// TIA Portal V16 export
// export: Created 2024-09-05T17:39:09.6685923Z, ExportSetting WithDefaults, DisplayName Totally Integrated Automation Portal, DisplayVersion V16 Update 6, DisplayName TIA Portal Version Control Interface, DisplayVersion V16 Update 2, DisplayName TIA Portal Openness, DisplayVersion V16 Update 6, DisplayName STEP 7 Professional, DisplayVersion V16 Update 6, DisplayName STEP 7 Safety, DisplayVersion V16, DisplayName WinCC Advanced, DisplayVersion V16 Update 6
DATA_BLOCK "CylinderGeneratedCalls_DB"   // DB51
VERSION : 0.1
// stored: AutoNumber true, DBAccessibleFromOPCUA true, InstanceOfName CylinderGeneratedCalls, InstanceOfType FB
"CylinderGeneratedCalls"
   // VAR
   //    MM2200_GrippingTubeFrontInstant { S7_SetPoint := 'True'} : "CylinderFaceplate";
   //    MM2201_GrippingTubeRearInstant { S7_SetPoint := 'True'} : "CylinderFaceplate";
   //    MM2220_HoldingSidememberInsideLeftInstant { S7_SetPoint := 'True'} : "CylinderFaceplate";
   //    MM2221_HoldingSidememberInsideRightInstant { S7_SetPoint := 'True'} : "CylinderFaceplate";
   //    MM2240_HoldingSidememberOutsideLeftInstant { S7_SetPoint := 'True'} : "CylinderFaceplate";
   //    MM2241_HoldingSidememberOutsideRightInstant { S7_SetPoint := 'True'} : "CylinderFaceplate";
   //    MM2500_GrippingTubeFrontInstant { S7_SetPoint := 'True'} : "CylinderFaceplate";
   //    MM2501_GrippingTubeRearInstant { S7_SetPoint := 'True'} : "CylinderFaceplate";
   //    MM2520_HoldingSidememberInsideLeftInstant { S7_SetPoint := 'True'} : "CylinderFaceplate";
   //    MM2521_HoldingSidememberInsideRightInstant { S7_SetPoint := 'True'} : "CylinderFaceplate";
   //    MM2540_HoldingSidememberOutsideLeftInstant { S7_SetPoint := 'True'} : "CylinderFaceplate";
   //    MM2541_HoldingSidememberOutsideRightInstant { S7_SetPoint := 'True'} : "CylinderFaceplate";
   //    MM300_ShiftingSupportRightInstant { S7_SetPoint := 'True'} : "CylinderFaceplate";
   //    MM302_ShiftingSupportLeftInstant { S7_SetPoint := 'True'} : "CylinderFaceplate";
   //    MM304_MovingStopRightInstant { S7_SetPoint := 'True'} : "CylinderFaceplate";
   //    MM306_MovingStopLeftInstant { S7_SetPoint := 'True'} : "CylinderFaceplate";
   //    MM340_RivetingUnitRightInstant { S7_SetPoint := 'True'} : "CylinderFaceplate";
   //    MM342_RivetingUnitLeftInstant { S7_SetPoint := 'True'} : "CylinderFaceplate";
   //    MM344_RivetingSupportRightInstant { S7_SetPoint := 'True'} : "CylinderFaceplate";
   //    MM346_RivetingSupportLeftInstant { S7_SetPoint := 'True'} : "CylinderFaceplate";
   //    MM350_ShiftWedgeRightInstant { S7_SetPoint := 'True'} : "CylinderFaceplate";
   //    MM352_ShiftWedgeLeftInstant { S7_SetPoint := 'True'} : "CylinderFaceplate";
   //    MM104_AutoejectGripperLiftingInstant { S7_SetPoint := 'True'} : "CylinderFaceplate";
   //    MM3100_SidememberSupportLeftInstant { S7_SetPoint := 'True'} : "CylinderFaceplate";
   //    MM3101_SidememberSupportRightInstant { S7_SetPoint := 'True'} : "CylinderFaceplate";
   // END_VAR
BEGIN
   MM2200_GrippingTubeFrontInstant.POWER_OK := TRUE;
   MM2200_GrippingTubeFrontInstant.CylinderNumber := 0;
   MM2200_GrippingTubeFrontInstant.HMICommand := 0;
   MM2200_GrippingTubeFrontInstant.BasicPositionCondition := TRUE;
   MM2200_GrippingTubeFrontInstant.WorkPositionCondition := FALSE;
   MM2200_GrippingTubeFrontInstant.BasicPositionSensor := TRUE;
   MM2200_GrippingTubeFrontInstant.WorkPositionSensor := FALSE;
   MM2200_GrippingTubeFrontInstant.TRIGGER := TRUE;
   MM2200_GrippingTubeFrontInstant.RESET := FALSE;
   MM2200_GrippingTubeFrontInstant.DELAY_BASIC := T#100MS;
   MM2200_GrippingTubeFrontInstant.DELAY_WORK := T#100MS;
   MM2200_GrippingTubeFrontInstant.DELAY_FREE := T#100MS;
   MM2200_GrippingTubeFrontInstant.ERROR_TIME := T#10S;
   MM2200_GrippingTubeFrontInstant.ValveDelay := T#0MS;
   MM2200_GrippingTubeFrontInstant.iNoCollisionBasic := TRUE;
   MM2200_GrippingTubeFrontInstant.iNoCollisionWork := TRUE;
   MM2200_GrippingTubeFrontInstant.iNoCollisionFree := TRUE;
   MM2200_GrippingTubeFrontInstant.VALVE_BASIC := TRUE;
   MM2200_GrippingTubeFrontInstant.VALVE_WORK := FALSE;
   MM2200_GrippingTubeFrontInstant.ERROR_BASIC := FALSE;
   MM2200_GrippingTubeFrontInstant.ERROR_WORK := FALSE;
   MM2200_GrippingTubeFrontInstant.HMIStatus := 257;
   MM2200_GrippingTubeFrontInstant.MOVE_BASIC := TRUE;
   MM2200_GrippingTubeFrontInstant.MOVE_WORK := FALSE;
   MM2200_GrippingTubeFrontInstant.MOVE_FREE := FALSE;
   MM2200_GrippingTubeFrontInstant."4l+Started" := FALSE;
   MM2200_GrippingTubeFrontInstant.InitCommandBP := FALSE;
   MM2200_GrippingTubeFrontInstant.InitCommandWP := FALSE;
   MM2200_GrippingTubeFrontInstant.BasicWorkStartWP := FALSE;
   MM2200_GrippingTubeFrontInstant.BasicWorkStartBP := FALSE;
   MM2200_GrippingTubeFrontInstant.work_valve := FALSE;
   MM2200_GrippingTubeFrontInstant.basic_valve := TRUE;
   MM2200_GrippingTubeFrontInstant.free_valve := FALSE;
   MM2200_GrippingTubeFrontInstant.baspos_error.PT := T#10S;
   MM2200_GrippingTubeFrontInstant.baspos_error.IN := FALSE;
   MM2200_GrippingTubeFrontInstant.workpos_error.PT := T#10S;
   MM2200_GrippingTubeFrontInstant.workpos_error.IN := FALSE;
   MM2200_GrippingTubeFrontInstant.baspos_delay.PT := T#100MS;
   MM2200_GrippingTubeFrontInstant.baspos_delay.IN := TRUE;
   MM2200_GrippingTubeFrontInstant.workpos_delay.PT := T#100MS;
   MM2200_GrippingTubeFrontInstant.workpos_delay.IN := FALSE;
   MM2200_GrippingTubeFrontInstant.CylinderOperationOld.InWp := FALSE;
   MM2200_GrippingTubeFrontInstant.CylinderOperationOld.InBp := TRUE;
   MM2200_GrippingTubeFrontInstant.CylinderOperationOld.InFp := FALSE;
   MM2200_GrippingTubeFrontInstant.CylinderOperationOld.ToWp := FALSE;
   MM2200_GrippingTubeFrontInstant.CylinderOperationOld.ToBp := TRUE;
   MM2200_GrippingTubeFrontInstant.CylinderOperationOld.ToFp := FALSE;
   MM2200_GrippingTubeFrontInstant.IEC_Timer_0_Instance.PT := T#0MS;
   MM2200_GrippingTubeFrontInstant.IEC_Timer_0_Instance.IN := FALSE;
   MM2200_GrippingTubeFrontInstant.R_TRIG_Instance.CLK := FALSE;
   MM2200_GrippingTubeFrontInstant.R_TRIG_Instance.Q := FALSE;
   MM2200_GrippingTubeFrontInstant.R_TRIG_Instance.Stat_Bit := FALSE;
   MM2200_GrippingTubeFrontInstant.IEC_Timer_0_Instance_1.PT := T#0MS;
   MM2200_GrippingTubeFrontInstant.IEC_Timer_0_Instance_1.IN := FALSE;
   MM2200_GrippingTubeFrontInstant.IEC_Timer_0_Instance_2.PT := T#0MS;
   MM2200_GrippingTubeFrontInstant.IEC_Timer_0_Instance_2.IN := FALSE;
   MM2200_GrippingTubeFrontInstant.IEC_Timer_0_Instance_3.PT := T#0MS;
   MM2200_GrippingTubeFrontInstant.IEC_Timer_0_Instance_3.IN := FALSE;
   MM2200_GrippingTubeFrontInstant.IEC_Timer_0_Instance_4.PT := T#0MS;
   MM2200_GrippingTubeFrontInstant.IEC_Timer_0_Instance_4.IN := TRUE;
   MM2201_GrippingTubeRearInstant.POWER_OK := TRUE;
   MM2201_GrippingTubeRearInstant.CylinderNumber := 1;
   MM2201_GrippingTubeRearInstant.HMICommand := 0;
   MM2201_GrippingTubeRearInstant.BasicPositionCondition := TRUE;
   MM2201_GrippingTubeRearInstant.WorkPositionCondition := FALSE;
   MM2201_GrippingTubeRearInstant.BasicPositionSensor := TRUE;
   MM2201_GrippingTubeRearInstant.WorkPositionSensor := FALSE;
   MM2201_GrippingTubeRearInstant.TRIGGER := TRUE;
   MM2201_GrippingTubeRearInstant.RESET := FALSE;
   MM2201_GrippingTubeRearInstant.DELAY_BASIC := T#100MS;
   MM2201_GrippingTubeRearInstant.DELAY_WORK := T#100MS;
   MM2201_GrippingTubeRearInstant.DELAY_FREE := T#100MS;
   MM2201_GrippingTubeRearInstant.ERROR_TIME := T#10S;
   MM2201_GrippingTubeRearInstant.ValveDelay := T#0MS;
   MM2201_GrippingTubeRearInstant.iNoCollisionBasic := TRUE;
   MM2201_GrippingTubeRearInstant.iNoCollisionWork := TRUE;
   MM2201_GrippingTubeRearInstant.iNoCollisionFree := TRUE;
   MM2201_GrippingTubeRearInstant.VALVE_BASIC := TRUE;
   MM2201_GrippingTubeRearInstant.VALVE_WORK := FALSE;
   MM2201_GrippingTubeRearInstant.ERROR_BASIC := FALSE;
   MM2201_GrippingTubeRearInstant.ERROR_WORK := FALSE;
   MM2201_GrippingTubeRearInstant.HMIStatus := 257;
   MM2201_GrippingTubeRearInstant.MOVE_BASIC := TRUE;
   MM2201_GrippingTubeRearInstant.MOVE_WORK := FALSE;
   MM2201_GrippingTubeRearInstant.MOVE_FREE := FALSE;
   MM2201_GrippingTubeRearInstant."4l+Started" := FALSE;
   MM2201_GrippingTubeRearInstant.InitCommandBP := FALSE;
   MM2201_GrippingTubeRearInstant.InitCommandWP := FALSE;
   MM2201_GrippingTubeRearInstant.BasicWorkStartWP := FALSE;
   MM2201_GrippingTubeRearInstant.BasicWorkStartBP := FALSE;
   MM2201_GrippingTubeRearInstant.work_valve := FALSE;
   MM2201_GrippingTubeRearInstant.basic_valve := TRUE;
   MM2201_GrippingTubeRearInstant.free_valve := FALSE;
   MM2201_GrippingTubeRearInstant.baspos_error.PT := T#10S;
   MM2201_GrippingTubeRearInstant.baspos_error.IN := FALSE;
   MM2201_GrippingTubeRearInstant.workpos_error.PT := T#10S;
   MM2201_GrippingTubeRearInstant.workpos_error.IN := FALSE;
   MM2201_GrippingTubeRearInstant.baspos_delay.PT := T#100MS;
   MM2201_GrippingTubeRearInstant.baspos_delay.IN := TRUE;
   MM2201_GrippingTubeRearInstant.workpos_delay.PT := T#100MS;
   MM2201_GrippingTubeRearInstant.workpos_delay.IN := FALSE;
   MM2201_GrippingTubeRearInstant.CylinderOperationOld.InWp := FALSE;
   MM2201_GrippingTubeRearInstant.CylinderOperationOld.InBp := TRUE;
   MM2201_GrippingTubeRearInstant.CylinderOperationOld.InFp := FALSE;
   MM2201_GrippingTubeRearInstant.CylinderOperationOld.ToWp := FALSE;
   MM2201_GrippingTubeRearInstant.CylinderOperationOld.ToBp := TRUE;
   MM2201_GrippingTubeRearInstant.CylinderOperationOld.ToFp := FALSE;
   MM2201_GrippingTubeRearInstant.IEC_Timer_0_Instance.PT := T#0MS;
   MM2201_GrippingTubeRearInstant.IEC_Timer_0_Instance.IN := FALSE;
   MM2201_GrippingTubeRearInstant.R_TRIG_Instance.CLK := FALSE;
   MM2201_GrippingTubeRearInstant.R_TRIG_Instance.Q := FALSE;
   MM2201_GrippingTubeRearInstant.R_TRIG_Instance.Stat_Bit := FALSE;
   MM2201_GrippingTubeRearInstant.IEC_Timer_0_Instance_1.PT := T#0MS;
   MM2201_GrippingTubeRearInstant.IEC_Timer_0_Instance_1.IN := FALSE;
   MM2201_GrippingTubeRearInstant.IEC_Timer_0_Instance_2.PT := T#0MS;
   MM2201_GrippingTubeRearInstant.IEC_Timer_0_Instance_2.IN := FALSE;
   MM2201_GrippingTubeRearInstant.IEC_Timer_0_Instance_3.PT := T#0MS;
   MM2201_GrippingTubeRearInstant.IEC_Timer_0_Instance_3.IN := FALSE;
   MM2201_GrippingTubeRearInstant.IEC_Timer_0_Instance_4.PT := T#0MS;
   MM2201_GrippingTubeRearInstant.IEC_Timer_0_Instance_4.IN := TRUE;
   MM2220_HoldingSidememberInsideLeftInstant.POWER_OK := TRUE;
   MM2220_HoldingSidememberInsideLeftInstant.CylinderNumber := 2;
   MM2220_HoldingSidememberInsideLeftInstant.HMICommand := 0;
   MM2220_HoldingSidememberInsideLeftInstant.BasicPositionCondition := TRUE;
   MM2220_HoldingSidememberInsideLeftInstant.WorkPositionCondition := FALSE;
   MM2220_HoldingSidememberInsideLeftInstant.BasicPositionSensor := TRUE;
   MM2220_HoldingSidememberInsideLeftInstant.WorkPositionSensor := FALSE;
   MM2220_HoldingSidememberInsideLeftInstant.TRIGGER := TRUE;
   MM2220_HoldingSidememberInsideLeftInstant.RESET := FALSE;
   MM2220_HoldingSidememberInsideLeftInstant.DELAY_BASIC := T#100MS;
   MM2220_HoldingSidememberInsideLeftInstant.DELAY_WORK := T#100MS;
   MM2220_HoldingSidememberInsideLeftInstant.DELAY_FREE := T#100MS;
   MM2220_HoldingSidememberInsideLeftInstant.ERROR_TIME := T#10S;
   MM2220_HoldingSidememberInsideLeftInstant.ValveDelay := T#0MS;
   MM2220_HoldingSidememberInsideLeftInstant.iNoCollisionBasic := TRUE;
   MM2220_HoldingSidememberInsideLeftInstant.iNoCollisionWork := TRUE;
   MM2220_HoldingSidememberInsideLeftInstant.iNoCollisionFree := TRUE;
   MM2220_HoldingSidememberInsideLeftInstant.VALVE_BASIC := TRUE;
   MM2220_HoldingSidememberInsideLeftInstant.VALVE_WORK := FALSE;
   MM2220_HoldingSidememberInsideLeftInstant.ERROR_BASIC := FALSE;
   MM2220_HoldingSidememberInsideLeftInstant.ERROR_WORK := FALSE;
   MM2220_HoldingSidememberInsideLeftInstant.HMIStatus := 257;
   MM2220_HoldingSidememberInsideLeftInstant.MOVE_BASIC := TRUE;
   MM2220_HoldingSidememberInsideLeftInstant.MOVE_WORK := FALSE;
   MM2220_HoldingSidememberInsideLeftInstant.MOVE_FREE := FALSE;
   MM2220_HoldingSidememberInsideLeftInstant."4l+Started" := FALSE;
   MM2220_HoldingSidememberInsideLeftInstant.InitCommandBP := FALSE;
   MM2220_HoldingSidememberInsideLeftInstant.InitCommandWP := FALSE;
   MM2220_HoldingSidememberInsideLeftInstant.BasicWorkStartWP := FALSE;
   MM2220_HoldingSidememberInsideLeftInstant.BasicWorkStartBP := FALSE;
   MM2220_HoldingSidememberInsideLeftInstant.work_valve := FALSE;
   MM2220_HoldingSidememberInsideLeftInstant.basic_valve := TRUE;
   MM2220_HoldingSidememberInsideLeftInstant.free_valve := FALSE;
   MM2220_HoldingSidememberInsideLeftInstant.baspos_error.PT := T#10S;
   MM2220_HoldingSidememberInsideLeftInstant.baspos_error.IN := FALSE;
   MM2220_HoldingSidememberInsideLeftInstant.workpos_error.PT := T#10S;
   MM2220_HoldingSidememberInsideLeftInstant.workpos_error.IN := FALSE;
   MM2220_HoldingSidememberInsideLeftInstant.baspos_delay.PT := T#100MS;
   MM2220_HoldingSidememberInsideLeftInstant.baspos_delay.IN := TRUE;
   MM2220_HoldingSidememberInsideLeftInstant.workpos_delay.PT := T#100MS;
   MM2220_HoldingSidememberInsideLeftInstant.workpos_delay.IN := FALSE;
   MM2220_HoldingSidememberInsideLeftInstant.CylinderOperationOld.InWp := FALSE;
   MM2220_HoldingSidememberInsideLeftInstant.CylinderOperationOld.InBp := TRUE;
   MM2220_HoldingSidememberInsideLeftInstant.CylinderOperationOld.InFp := FALSE;
   MM2220_HoldingSidememberInsideLeftInstant.CylinderOperationOld.ToWp := FALSE;
   MM2220_HoldingSidememberInsideLeftInstant.CylinderOperationOld.ToBp := TRUE;
   MM2220_HoldingSidememberInsideLeftInstant.CylinderOperationOld.ToFp := FALSE;
   MM2220_HoldingSidememberInsideLeftInstant.IEC_Timer_0_Instance.PT := T#0MS;
   MM2220_HoldingSidememberInsideLeftInstant.IEC_Timer_0_Instance.IN := FALSE;
   MM2220_HoldingSidememberInsideLeftInstant.R_TRIG_Instance.CLK := FALSE;
   MM2220_HoldingSidememberInsideLeftInstant.R_TRIG_Instance.Q := FALSE;
   MM2220_HoldingSidememberInsideLeftInstant.R_TRIG_Instance.Stat_Bit := FALSE;
   MM2220_HoldingSidememberInsideLeftInstant.IEC_Timer_0_Instance_1.PT := T#0MS;
   MM2220_HoldingSidememberInsideLeftInstant.IEC_Timer_0_Instance_1.IN := FALSE;
   MM2220_HoldingSidememberInsideLeftInstant.IEC_Timer_0_Instance_2.PT := T#0MS;
   MM2220_HoldingSidememberInsideLeftInstant.IEC_Timer_0_Instance_2.IN := FALSE;
   MM2220_HoldingSidememberInsideLeftInstant.IEC_Timer_0_Instance_3.PT := T#0MS;
   MM2220_HoldingSidememberInsideLeftInstant.IEC_Timer_0_Instance_3.IN := FALSE;
   MM2220_HoldingSidememberInsideLeftInstant.IEC_Timer_0_Instance_4.PT := T#0MS;
   MM2220_HoldingSidememberInsideLeftInstant.IEC_Timer_0_Instance_4.IN := TRUE;
   MM2221_HoldingSidememberInsideRightInstant.POWER_OK := TRUE;
   MM2221_HoldingSidememberInsideRightInstant.CylinderNumber := 3;
   MM2221_HoldingSidememberInsideRightInstant.HMICommand := 0;
   MM2221_HoldingSidememberInsideRightInstant.BasicPositionCondition := TRUE;
   MM2221_HoldingSidememberInsideRightInstant.WorkPositionCondition := FALSE;
   MM2221_HoldingSidememberInsideRightInstant.BasicPositionSensor := TRUE;
   MM2221_HoldingSidememberInsideRightInstant.WorkPositionSensor := FALSE;
   MM2221_HoldingSidememberInsideRightInstant.TRIGGER := TRUE;
   MM2221_HoldingSidememberInsideRightInstant.RESET := FALSE;
   MM2221_HoldingSidememberInsideRightInstant.DELAY_BASIC := T#100MS;
   MM2221_HoldingSidememberInsideRightInstant.DELAY_WORK := T#100MS;
   MM2221_HoldingSidememberInsideRightInstant.DELAY_FREE := T#100MS;
   MM2221_HoldingSidememberInsideRightInstant.ERROR_TIME := T#10S;
   MM2221_HoldingSidememberInsideRightInstant.ValveDelay := T#0MS;
   MM2221_HoldingSidememberInsideRightInstant.iNoCollisionBasic := TRUE;
   MM2221_HoldingSidememberInsideRightInstant.iNoCollisionWork := TRUE;
   MM2221_HoldingSidememberInsideRightInstant.iNoCollisionFree := TRUE;
   MM2221_HoldingSidememberInsideRightInstant.VALVE_BASIC := TRUE;
   MM2221_HoldingSidememberInsideRightInstant.VALVE_WORK := FALSE;
   MM2221_HoldingSidememberInsideRightInstant.ERROR_BASIC := FALSE;
   MM2221_HoldingSidememberInsideRightInstant.ERROR_WORK := FALSE;
   MM2221_HoldingSidememberInsideRightInstant.HMIStatus := 257;
   MM2221_HoldingSidememberInsideRightInstant.MOVE_BASIC := TRUE;
   MM2221_HoldingSidememberInsideRightInstant.MOVE_WORK := FALSE;
   MM2221_HoldingSidememberInsideRightInstant.MOVE_FREE := FALSE;
   MM2221_HoldingSidememberInsideRightInstant."4l+Started" := FALSE;
   MM2221_HoldingSidememberInsideRightInstant.InitCommandBP := FALSE;
   MM2221_HoldingSidememberInsideRightInstant.InitCommandWP := FALSE;
   MM2221_HoldingSidememberInsideRightInstant.BasicWorkStartWP := FALSE;
   MM2221_HoldingSidememberInsideRightInstant.BasicWorkStartBP := FALSE;
   MM2221_HoldingSidememberInsideRightInstant.work_valve := FALSE;
   MM2221_HoldingSidememberInsideRightInstant.basic_valve := TRUE;
   MM2221_HoldingSidememberInsideRightInstant.free_valve := FALSE;
   MM2221_HoldingSidememberInsideRightInstant.baspos_error.PT := T#10S;
   MM2221_HoldingSidememberInsideRightInstant.baspos_error.IN := FALSE;
   MM2221_HoldingSidememberInsideRightInstant.workpos_error.PT := T#10S;
   MM2221_HoldingSidememberInsideRightInstant.workpos_error.IN := FALSE;
   MM2221_HoldingSidememberInsideRightInstant.baspos_delay.PT := T#100MS;
   MM2221_HoldingSidememberInsideRightInstant.baspos_delay.IN := TRUE;
   MM2221_HoldingSidememberInsideRightInstant.workpos_delay.PT := T#100MS;
   MM2221_HoldingSidememberInsideRightInstant.workpos_delay.IN := FALSE;
   MM2221_HoldingSidememberInsideRightInstant.CylinderOperationOld.InWp := FALSE;
   MM2221_HoldingSidememberInsideRightInstant.CylinderOperationOld.InBp := TRUE;
   MM2221_HoldingSidememberInsideRightInstant.CylinderOperationOld.InFp := FALSE;
   MM2221_HoldingSidememberInsideRightInstant.CylinderOperationOld.ToWp := FALSE;
   MM2221_HoldingSidememberInsideRightInstant.CylinderOperationOld.ToBp := TRUE;
   MM2221_HoldingSidememberInsideRightInstant.CylinderOperationOld.ToFp := FALSE;
   MM2221_HoldingSidememberInsideRightInstant.IEC_Timer_0_Instance.PT := T#0MS;
   MM2221_HoldingSidememberInsideRightInstant.IEC_Timer_0_Instance.IN := FALSE;
   MM2221_HoldingSidememberInsideRightInstant.R_TRIG_Instance.CLK := FALSE;
   MM2221_HoldingSidememberInsideRightInstant.R_TRIG_Instance.Q := FALSE;
   MM2221_HoldingSidememberInsideRightInstant.R_TRIG_Instance.Stat_Bit := FALSE;
   MM2221_HoldingSidememberInsideRightInstant.IEC_Timer_0_Instance_1.PT := T#0MS;
   MM2221_HoldingSidememberInsideRightInstant.IEC_Timer_0_Instance_1.IN := FALSE;
   MM2221_HoldingSidememberInsideRightInstant.IEC_Timer_0_Instance_2.PT := T#0MS;
   MM2221_HoldingSidememberInsideRightInstant.IEC_Timer_0_Instance_2.IN := FALSE;
   MM2221_HoldingSidememberInsideRightInstant.IEC_Timer_0_Instance_3.PT := T#0MS;
   MM2221_HoldingSidememberInsideRightInstant.IEC_Timer_0_Instance_3.IN := FALSE;
   MM2221_HoldingSidememberInsideRightInstant.IEC_Timer_0_Instance_4.PT := T#0MS;
   MM2221_HoldingSidememberInsideRightInstant.IEC_Timer_0_Instance_4.IN := TRUE;
   MM2240_HoldingSidememberOutsideLeftInstant.POWER_OK := TRUE;
   MM2240_HoldingSidememberOutsideLeftInstant.CylinderNumber := 4;
   MM2240_HoldingSidememberOutsideLeftInstant.HMICommand := 0;
   MM2240_HoldingSidememberOutsideLeftInstant.BasicPositionCondition := TRUE;
   MM2240_HoldingSidememberOutsideLeftInstant.WorkPositionCondition := FALSE;
   MM2240_HoldingSidememberOutsideLeftInstant.BasicPositionSensor := TRUE;
   MM2240_HoldingSidememberOutsideLeftInstant.WorkPositionSensor := FALSE;
   MM2240_HoldingSidememberOutsideLeftInstant.TRIGGER := TRUE;
   MM2240_HoldingSidememberOutsideLeftInstant.RESET := FALSE;
   MM2240_HoldingSidememberOutsideLeftInstant.DELAY_BASIC := T#100MS;
   MM2240_HoldingSidememberOutsideLeftInstant.DELAY_WORK := T#100MS;
   MM2240_HoldingSidememberOutsideLeftInstant.DELAY_FREE := T#100MS;
   MM2240_HoldingSidememberOutsideLeftInstant.ERROR_TIME := T#10S;
   MM2240_HoldingSidememberOutsideLeftInstant.ValveDelay := T#0MS;
   MM2240_HoldingSidememberOutsideLeftInstant.iNoCollisionBasic := TRUE;
   MM2240_HoldingSidememberOutsideLeftInstant.iNoCollisionWork := TRUE;
   MM2240_HoldingSidememberOutsideLeftInstant.iNoCollisionFree := TRUE;
   MM2240_HoldingSidememberOutsideLeftInstant.VALVE_BASIC := TRUE;
   MM2240_HoldingSidememberOutsideLeftInstant.VALVE_WORK := FALSE;
   MM2240_HoldingSidememberOutsideLeftInstant.ERROR_BASIC := FALSE;
   MM2240_HoldingSidememberOutsideLeftInstant.ERROR_WORK := FALSE;
   MM2240_HoldingSidememberOutsideLeftInstant.HMIStatus := 257;
   MM2240_HoldingSidememberOutsideLeftInstant.MOVE_BASIC := TRUE;
   MM2240_HoldingSidememberOutsideLeftInstant.MOVE_WORK := FALSE;
   MM2240_HoldingSidememberOutsideLeftInstant.MOVE_FREE := FALSE;
   MM2240_HoldingSidememberOutsideLeftInstant."4l+Started" := FALSE;
   MM2240_HoldingSidememberOutsideLeftInstant.InitCommandBP := FALSE;
   MM2240_HoldingSidememberOutsideLeftInstant.InitCommandWP := FALSE;
   MM2240_HoldingSidememberOutsideLeftInstant.BasicWorkStartWP := FALSE;
   MM2240_HoldingSidememberOutsideLeftInstant.BasicWorkStartBP := FALSE;
   MM2240_HoldingSidememberOutsideLeftInstant.work_valve := FALSE;
   MM2240_HoldingSidememberOutsideLeftInstant.basic_valve := TRUE;
   MM2240_HoldingSidememberOutsideLeftInstant.free_valve := FALSE;
   MM2240_HoldingSidememberOutsideLeftInstant.baspos_error.PT := T#10S;
   MM2240_HoldingSidememberOutsideLeftInstant.baspos_error.IN := FALSE;
   MM2240_HoldingSidememberOutsideLeftInstant.workpos_error.PT := T#10S;
   MM2240_HoldingSidememberOutsideLeftInstant.workpos_error.IN := FALSE;
   MM2240_HoldingSidememberOutsideLeftInstant.baspos_delay.PT := T#100MS;
   MM2240_HoldingSidememberOutsideLeftInstant.baspos_delay.IN := TRUE;
   MM2240_HoldingSidememberOutsideLeftInstant.workpos_delay.PT := T#100MS;
   MM2240_HoldingSidememberOutsideLeftInstant.workpos_delay.IN := FALSE;
   MM2240_HoldingSidememberOutsideLeftInstant.CylinderOperationOld.InWp := FALSE;
   MM2240_HoldingSidememberOutsideLeftInstant.CylinderOperationOld.InBp := TRUE;
   MM2240_HoldingSidememberOutsideLeftInstant.CylinderOperationOld.InFp := FALSE;
   MM2240_HoldingSidememberOutsideLeftInstant.CylinderOperationOld.ToWp := FALSE;
   MM2240_HoldingSidememberOutsideLeftInstant.CylinderOperationOld.ToBp := TRUE;
   MM2240_HoldingSidememberOutsideLeftInstant.CylinderOperationOld.ToFp := FALSE;
   MM2240_HoldingSidememberOutsideLeftInstant.IEC_Timer_0_Instance.PT := T#0MS;
   MM2240_HoldingSidememberOutsideLeftInstant.IEC_Timer_0_Instance.IN := FALSE;
   MM2240_HoldingSidememberOutsideLeftInstant.R_TRIG_Instance.CLK := FALSE;
   MM2240_HoldingSidememberOutsideLeftInstant.R_TRIG_Instance.Q := FALSE;
   MM2240_HoldingSidememberOutsideLeftInstant.R_TRIG_Instance.Stat_Bit := FALSE;
   MM2240_HoldingSidememberOutsideLeftInstant.IEC_Timer_0_Instance_1.PT := T#0MS;
   MM2240_HoldingSidememberOutsideLeftInstant.IEC_Timer_0_Instance_1.IN := FALSE;
   MM2240_HoldingSidememberOutsideLeftInstant.IEC_Timer_0_Instance_2.PT := T#0MS;
   MM2240_HoldingSidememberOutsideLeftInstant.IEC_Timer_0_Instance_2.IN := FALSE;
   MM2240_HoldingSidememberOutsideLeftInstant.IEC_Timer_0_Instance_3.PT := T#0MS;
   MM2240_HoldingSidememberOutsideLeftInstant.IEC_Timer_0_Instance_3.IN := FALSE;
   MM2240_HoldingSidememberOutsideLeftInstant.IEC_Timer_0_Instance_4.PT := T#0MS;
   MM2240_HoldingSidememberOutsideLeftInstant.IEC_Timer_0_Instance_4.IN := TRUE;
   MM2241_HoldingSidememberOutsideRightInstant.POWER_OK := TRUE;
   MM2241_HoldingSidememberOutsideRightInstant.CylinderNumber := 5;
   MM2241_HoldingSidememberOutsideRightInstant.HMICommand := 0;
   MM2241_HoldingSidememberOutsideRightInstant.BasicPositionCondition := TRUE;
   MM2241_HoldingSidememberOutsideRightInstant.WorkPositionCondition := FALSE;
   MM2241_HoldingSidememberOutsideRightInstant.BasicPositionSensor := TRUE;
   MM2241_HoldingSidememberOutsideRightInstant.WorkPositionSensor := FALSE;
   MM2241_HoldingSidememberOutsideRightInstant.TRIGGER := TRUE;
   MM2241_HoldingSidememberOutsideRightInstant.RESET := FALSE;
   MM2241_HoldingSidememberOutsideRightInstant.DELAY_BASIC := T#100MS;
   MM2241_HoldingSidememberOutsideRightInstant.DELAY_WORK := T#100MS;
   MM2241_HoldingSidememberOutsideRightInstant.DELAY_FREE := T#100MS;
   MM2241_HoldingSidememberOutsideRightInstant.ERROR_TIME := T#10S;
   MM2241_HoldingSidememberOutsideRightInstant.ValveDelay := T#0MS;
   MM2241_HoldingSidememberOutsideRightInstant.iNoCollisionBasic := TRUE;
   MM2241_HoldingSidememberOutsideRightInstant.iNoCollisionWork := TRUE;
   MM2241_HoldingSidememberOutsideRightInstant.iNoCollisionFree := TRUE;
   MM2241_HoldingSidememberOutsideRightInstant.VALVE_BASIC := FALSE;
   MM2241_HoldingSidememberOutsideRightInstant.VALVE_WORK := FALSE;
   MM2241_HoldingSidememberOutsideRightInstant.ERROR_BASIC := FALSE;
   MM2241_HoldingSidememberOutsideRightInstant.ERROR_WORK := FALSE;
   MM2241_HoldingSidememberOutsideRightInstant.HMIStatus := 1;
   MM2241_HoldingSidememberOutsideRightInstant.MOVE_BASIC := FALSE;
   MM2241_HoldingSidememberOutsideRightInstant.MOVE_WORK := FALSE;
   MM2241_HoldingSidememberOutsideRightInstant.MOVE_FREE := TRUE;
   MM2241_HoldingSidememberOutsideRightInstant."4l+Started" := FALSE;
   MM2241_HoldingSidememberOutsideRightInstant.InitCommandBP := FALSE;
   MM2241_HoldingSidememberOutsideRightInstant.InitCommandWP := FALSE;
   MM2241_HoldingSidememberOutsideRightInstant.BasicWorkStartWP := FALSE;
   MM2241_HoldingSidememberOutsideRightInstant.BasicWorkStartBP := FALSE;
   MM2241_HoldingSidememberOutsideRightInstant.work_valve := FALSE;
   MM2241_HoldingSidememberOutsideRightInstant.basic_valve := FALSE;
   MM2241_HoldingSidememberOutsideRightInstant.free_valve := FALSE;
   MM2241_HoldingSidememberOutsideRightInstant.baspos_error.PT := T#10S;
   MM2241_HoldingSidememberOutsideRightInstant.baspos_error.IN := FALSE;
   MM2241_HoldingSidememberOutsideRightInstant.workpos_error.PT := T#10S;
   MM2241_HoldingSidememberOutsideRightInstant.workpos_error.IN := FALSE;
   MM2241_HoldingSidememberOutsideRightInstant.baspos_delay.PT := T#100MS;
   MM2241_HoldingSidememberOutsideRightInstant.baspos_delay.IN := FALSE;
   MM2241_HoldingSidememberOutsideRightInstant.workpos_delay.PT := T#100MS;
   MM2241_HoldingSidememberOutsideRightInstant.workpos_delay.IN := FALSE;
   MM2241_HoldingSidememberOutsideRightInstant.CylinderOperationOld.InWp := FALSE;
   MM2241_HoldingSidememberOutsideRightInstant.CylinderOperationOld.InBp := TRUE;
   MM2241_HoldingSidememberOutsideRightInstant.CylinderOperationOld.InFp := TRUE;
   MM2241_HoldingSidememberOutsideRightInstant.CylinderOperationOld.ToWp := FALSE;
   MM2241_HoldingSidememberOutsideRightInstant.CylinderOperationOld.ToBp := FALSE;
   MM2241_HoldingSidememberOutsideRightInstant.CylinderOperationOld.ToFp := TRUE;
   MM2241_HoldingSidememberOutsideRightInstant.IEC_Timer_0_Instance.PT := T#0MS;
   MM2241_HoldingSidememberOutsideRightInstant.IEC_Timer_0_Instance.IN := FALSE;
   MM2241_HoldingSidememberOutsideRightInstant.R_TRIG_Instance.CLK := FALSE;
   MM2241_HoldingSidememberOutsideRightInstant.R_TRIG_Instance.Q := FALSE;
   MM2241_HoldingSidememberOutsideRightInstant.R_TRIG_Instance.Stat_Bit := FALSE;
   MM2241_HoldingSidememberOutsideRightInstant.IEC_Timer_0_Instance_1.PT := T#0MS;
   MM2241_HoldingSidememberOutsideRightInstant.IEC_Timer_0_Instance_1.IN := FALSE;
   MM2241_HoldingSidememberOutsideRightInstant.IEC_Timer_0_Instance_2.PT := T#0MS;
   MM2241_HoldingSidememberOutsideRightInstant.IEC_Timer_0_Instance_2.IN := FALSE;
   MM2241_HoldingSidememberOutsideRightInstant.IEC_Timer_0_Instance_3.PT := T#0MS;
   MM2241_HoldingSidememberOutsideRightInstant.IEC_Timer_0_Instance_3.IN := FALSE;
   MM2241_HoldingSidememberOutsideRightInstant.IEC_Timer_0_Instance_4.PT := T#0MS;
   MM2241_HoldingSidememberOutsideRightInstant.IEC_Timer_0_Instance_4.IN := FALSE;
   MM2500_GrippingTubeFrontInstant.POWER_OK := TRUE;
   MM2500_GrippingTubeFrontInstant.CylinderNumber := 6;
   MM2500_GrippingTubeFrontInstant.HMICommand := 0;
   MM2500_GrippingTubeFrontInstant.BasicPositionCondition := TRUE;
   MM2500_GrippingTubeFrontInstant.WorkPositionCondition := FALSE;
   MM2500_GrippingTubeFrontInstant.BasicPositionSensor := TRUE;
   MM2500_GrippingTubeFrontInstant.WorkPositionSensor := FALSE;
   MM2500_GrippingTubeFrontInstant.TRIGGER := TRUE;
   MM2500_GrippingTubeFrontInstant.RESET := FALSE;
   MM2500_GrippingTubeFrontInstant.DELAY_BASIC := T#100MS;
   MM2500_GrippingTubeFrontInstant.DELAY_WORK := T#100MS;
   MM2500_GrippingTubeFrontInstant.DELAY_FREE := T#100MS;
   MM2500_GrippingTubeFrontInstant.ERROR_TIME := T#10S;
   MM2500_GrippingTubeFrontInstant.ValveDelay := T#0MS;
   MM2500_GrippingTubeFrontInstant.iNoCollisionBasic := TRUE;
   MM2500_GrippingTubeFrontInstant.iNoCollisionWork := TRUE;
   MM2500_GrippingTubeFrontInstant.iNoCollisionFree := TRUE;
   MM2500_GrippingTubeFrontInstant.VALVE_BASIC := FALSE;
   MM2500_GrippingTubeFrontInstant.VALVE_WORK := FALSE;
   MM2500_GrippingTubeFrontInstant.ERROR_BASIC := FALSE;
   MM2500_GrippingTubeFrontInstant.ERROR_WORK := FALSE;
   MM2500_GrippingTubeFrontInstant.HMIStatus := 1;
   MM2500_GrippingTubeFrontInstant.MOVE_BASIC := FALSE;
   MM2500_GrippingTubeFrontInstant.MOVE_WORK := FALSE;
   MM2500_GrippingTubeFrontInstant.MOVE_FREE := TRUE;
   MM2500_GrippingTubeFrontInstant."4l+Started" := FALSE;
   MM2500_GrippingTubeFrontInstant.InitCommandBP := FALSE;
   MM2500_GrippingTubeFrontInstant.InitCommandWP := FALSE;
   MM2500_GrippingTubeFrontInstant.BasicWorkStartWP := FALSE;
   MM2500_GrippingTubeFrontInstant.BasicWorkStartBP := FALSE;
   MM2500_GrippingTubeFrontInstant.work_valve := FALSE;
   MM2500_GrippingTubeFrontInstant.basic_valve := FALSE;
   MM2500_GrippingTubeFrontInstant.free_valve := FALSE;
   MM2500_GrippingTubeFrontInstant.baspos_error.PT := T#10S;
   MM2500_GrippingTubeFrontInstant.baspos_error.IN := FALSE;
   MM2500_GrippingTubeFrontInstant.workpos_error.PT := T#10S;
   MM2500_GrippingTubeFrontInstant.workpos_error.IN := FALSE;
   MM2500_GrippingTubeFrontInstant.baspos_delay.PT := T#100MS;
   MM2500_GrippingTubeFrontInstant.baspos_delay.IN := FALSE;
   MM2500_GrippingTubeFrontInstant.workpos_delay.PT := T#100MS;
   MM2500_GrippingTubeFrontInstant.workpos_delay.IN := FALSE;
   MM2500_GrippingTubeFrontInstant.CylinderOperationOld.InWp := FALSE;
   MM2500_GrippingTubeFrontInstant.CylinderOperationOld.InBp := TRUE;
   MM2500_GrippingTubeFrontInstant.CylinderOperationOld.InFp := TRUE;
   MM2500_GrippingTubeFrontInstant.CylinderOperationOld.ToWp := FALSE;
   MM2500_GrippingTubeFrontInstant.CylinderOperationOld.ToBp := FALSE;
   MM2500_GrippingTubeFrontInstant.CylinderOperationOld.ToFp := TRUE;
   MM2500_GrippingTubeFrontInstant.IEC_Timer_0_Instance.PT := T#0MS;
   MM2500_GrippingTubeFrontInstant.IEC_Timer_0_Instance.IN := FALSE;
   MM2500_GrippingTubeFrontInstant.R_TRIG_Instance.CLK := FALSE;
   MM2500_GrippingTubeFrontInstant.R_TRIG_Instance.Q := FALSE;
   MM2500_GrippingTubeFrontInstant.R_TRIG_Instance.Stat_Bit := FALSE;
   MM2500_GrippingTubeFrontInstant.IEC_Timer_0_Instance_1.PT := T#0MS;
   MM2500_GrippingTubeFrontInstant.IEC_Timer_0_Instance_1.IN := FALSE;
   MM2500_GrippingTubeFrontInstant.IEC_Timer_0_Instance_2.PT := T#0MS;
   MM2500_GrippingTubeFrontInstant.IEC_Timer_0_Instance_2.IN := FALSE;
   MM2500_GrippingTubeFrontInstant.IEC_Timer_0_Instance_3.PT := T#0MS;
   MM2500_GrippingTubeFrontInstant.IEC_Timer_0_Instance_3.IN := FALSE;
   MM2500_GrippingTubeFrontInstant.IEC_Timer_0_Instance_4.PT := T#0MS;
   MM2500_GrippingTubeFrontInstant.IEC_Timer_0_Instance_4.IN := FALSE;
   MM2501_GrippingTubeRearInstant.POWER_OK := TRUE;
   MM2501_GrippingTubeRearInstant.CylinderNumber := 7;
   MM2501_GrippingTubeRearInstant.HMICommand := 0;
   MM2501_GrippingTubeRearInstant.BasicPositionCondition := TRUE;
   MM2501_GrippingTubeRearInstant.WorkPositionCondition := FALSE;
   MM2501_GrippingTubeRearInstant.BasicPositionSensor := TRUE;
   MM2501_GrippingTubeRearInstant.WorkPositionSensor := FALSE;
   MM2501_GrippingTubeRearInstant.TRIGGER := TRUE;
   MM2501_GrippingTubeRearInstant.RESET := FALSE;
   MM2501_GrippingTubeRearInstant.DELAY_BASIC := T#100MS;
   MM2501_GrippingTubeRearInstant.DELAY_WORK := T#100MS;
   MM2501_GrippingTubeRearInstant.DELAY_FREE := T#100MS;
   MM2501_GrippingTubeRearInstant.ERROR_TIME := T#10S;
   MM2501_GrippingTubeRearInstant.ValveDelay := T#0MS;
   MM2501_GrippingTubeRearInstant.iNoCollisionBasic := TRUE;
   MM2501_GrippingTubeRearInstant.iNoCollisionWork := TRUE;
   MM2501_GrippingTubeRearInstant.iNoCollisionFree := TRUE;
   MM2501_GrippingTubeRearInstant.VALVE_BASIC := TRUE;
   MM2501_GrippingTubeRearInstant.VALVE_WORK := FALSE;
   MM2501_GrippingTubeRearInstant.ERROR_BASIC := FALSE;
   MM2501_GrippingTubeRearInstant.ERROR_WORK := FALSE;
   MM2501_GrippingTubeRearInstant.HMIStatus := 257;
   MM2501_GrippingTubeRearInstant.MOVE_BASIC := TRUE;
   MM2501_GrippingTubeRearInstant.MOVE_WORK := FALSE;
   MM2501_GrippingTubeRearInstant.MOVE_FREE := FALSE;
   MM2501_GrippingTubeRearInstant."4l+Started" := FALSE;
   MM2501_GrippingTubeRearInstant.InitCommandBP := FALSE;
   MM2501_GrippingTubeRearInstant.InitCommandWP := FALSE;
   MM2501_GrippingTubeRearInstant.BasicWorkStartWP := FALSE;
   MM2501_GrippingTubeRearInstant.BasicWorkStartBP := FALSE;
   MM2501_GrippingTubeRearInstant.work_valve := FALSE;
   MM2501_GrippingTubeRearInstant.basic_valve := TRUE;
   MM2501_GrippingTubeRearInstant.free_valve := FALSE;
   MM2501_GrippingTubeRearInstant.baspos_error.PT := T#10S;
   MM2501_GrippingTubeRearInstant.baspos_error.IN := FALSE;
   MM2501_GrippingTubeRearInstant.workpos_error.PT := T#10S;
   MM2501_GrippingTubeRearInstant.workpos_error.IN := FALSE;
   MM2501_GrippingTubeRearInstant.baspos_delay.PT := T#100MS;
   MM2501_GrippingTubeRearInstant.baspos_delay.IN := TRUE;
   MM2501_GrippingTubeRearInstant.workpos_delay.PT := T#100MS;
   MM2501_GrippingTubeRearInstant.workpos_delay.IN := FALSE;
   MM2501_GrippingTubeRearInstant.CylinderOperationOld.InWp := FALSE;
   MM2501_GrippingTubeRearInstant.CylinderOperationOld.InBp := TRUE;
   MM2501_GrippingTubeRearInstant.CylinderOperationOld.InFp := FALSE;
   MM2501_GrippingTubeRearInstant.CylinderOperationOld.ToWp := FALSE;
   MM2501_GrippingTubeRearInstant.CylinderOperationOld.ToBp := TRUE;
   MM2501_GrippingTubeRearInstant.CylinderOperationOld.ToFp := FALSE;
   MM2501_GrippingTubeRearInstant.IEC_Timer_0_Instance.PT := T#0MS;
   MM2501_GrippingTubeRearInstant.IEC_Timer_0_Instance.IN := FALSE;
   MM2501_GrippingTubeRearInstant.R_TRIG_Instance.CLK := FALSE;
   MM2501_GrippingTubeRearInstant.R_TRIG_Instance.Q := FALSE;
   MM2501_GrippingTubeRearInstant.R_TRIG_Instance.Stat_Bit := FALSE;
   MM2501_GrippingTubeRearInstant.IEC_Timer_0_Instance_1.PT := T#0MS;
   MM2501_GrippingTubeRearInstant.IEC_Timer_0_Instance_1.IN := FALSE;
   MM2501_GrippingTubeRearInstant.IEC_Timer_0_Instance_2.PT := T#0MS;
   MM2501_GrippingTubeRearInstant.IEC_Timer_0_Instance_2.IN := FALSE;
   MM2501_GrippingTubeRearInstant.IEC_Timer_0_Instance_3.PT := T#0MS;
   MM2501_GrippingTubeRearInstant.IEC_Timer_0_Instance_3.IN := FALSE;
   MM2501_GrippingTubeRearInstant.IEC_Timer_0_Instance_4.PT := T#0MS;
   MM2501_GrippingTubeRearInstant.IEC_Timer_0_Instance_4.IN := TRUE;
   MM2520_HoldingSidememberInsideLeftInstant.POWER_OK := TRUE;
   MM2520_HoldingSidememberInsideLeftInstant.CylinderNumber := 8;
   MM2520_HoldingSidememberInsideLeftInstant.HMICommand := 0;
   MM2520_HoldingSidememberInsideLeftInstant.BasicPositionCondition := TRUE;
   MM2520_HoldingSidememberInsideLeftInstant.WorkPositionCondition := FALSE;
   MM2520_HoldingSidememberInsideLeftInstant.BasicPositionSensor := TRUE;
   MM2520_HoldingSidememberInsideLeftInstant.WorkPositionSensor := FALSE;
   MM2520_HoldingSidememberInsideLeftInstant.TRIGGER := TRUE;
   MM2520_HoldingSidememberInsideLeftInstant.RESET := FALSE;
   MM2520_HoldingSidememberInsideLeftInstant.DELAY_BASIC := T#100MS;
   MM2520_HoldingSidememberInsideLeftInstant.DELAY_WORK := T#100MS;
   MM2520_HoldingSidememberInsideLeftInstant.DELAY_FREE := T#100MS;
   MM2520_HoldingSidememberInsideLeftInstant.ERROR_TIME := T#10S;
   MM2520_HoldingSidememberInsideLeftInstant.ValveDelay := T#0MS;
   MM2520_HoldingSidememberInsideLeftInstant.iNoCollisionBasic := TRUE;
   MM2520_HoldingSidememberInsideLeftInstant.iNoCollisionWork := TRUE;
   MM2520_HoldingSidememberInsideLeftInstant.iNoCollisionFree := TRUE;
   MM2520_HoldingSidememberInsideLeftInstant.VALVE_BASIC := TRUE;
   MM2520_HoldingSidememberInsideLeftInstant.VALVE_WORK := FALSE;
   MM2520_HoldingSidememberInsideLeftInstant.ERROR_BASIC := FALSE;
   MM2520_HoldingSidememberInsideLeftInstant.ERROR_WORK := FALSE;
   MM2520_HoldingSidememberInsideLeftInstant.HMIStatus := 257;
   MM2520_HoldingSidememberInsideLeftInstant.MOVE_BASIC := TRUE;
   MM2520_HoldingSidememberInsideLeftInstant.MOVE_WORK := FALSE;
   MM2520_HoldingSidememberInsideLeftInstant.MOVE_FREE := FALSE;
   MM2520_HoldingSidememberInsideLeftInstant."4l+Started" := FALSE;
   MM2520_HoldingSidememberInsideLeftInstant.InitCommandBP := FALSE;
   MM2520_HoldingSidememberInsideLeftInstant.InitCommandWP := FALSE;
   MM2520_HoldingSidememberInsideLeftInstant.BasicWorkStartWP := FALSE;
   MM2520_HoldingSidememberInsideLeftInstant.BasicWorkStartBP := FALSE;
   MM2520_HoldingSidememberInsideLeftInstant.work_valve := FALSE;
   MM2520_HoldingSidememberInsideLeftInstant.basic_valve := TRUE;
   MM2520_HoldingSidememberInsideLeftInstant.free_valve := FALSE;
   MM2520_HoldingSidememberInsideLeftInstant.baspos_error.PT := T#10S;
   MM2520_HoldingSidememberInsideLeftInstant.baspos_error.IN := FALSE;
   MM2520_HoldingSidememberInsideLeftInstant.workpos_error.PT := T#10S;
   MM2520_HoldingSidememberInsideLeftInstant.workpos_error.IN := FALSE;
   MM2520_HoldingSidememberInsideLeftInstant.baspos_delay.PT := T#100MS;
   MM2520_HoldingSidememberInsideLeftInstant.baspos_delay.IN := TRUE;
   MM2520_HoldingSidememberInsideLeftInstant.workpos_delay.PT := T#100MS;
   MM2520_HoldingSidememberInsideLeftInstant.workpos_delay.IN := FALSE;
   MM2520_HoldingSidememberInsideLeftInstant.CylinderOperationOld.InWp := FALSE;
   MM2520_HoldingSidememberInsideLeftInstant.CylinderOperationOld.InBp := TRUE;
   MM2520_HoldingSidememberInsideLeftInstant.CylinderOperationOld.InFp := FALSE;
   MM2520_HoldingSidememberInsideLeftInstant.CylinderOperationOld.ToWp := FALSE;
   MM2520_HoldingSidememberInsideLeftInstant.CylinderOperationOld.ToBp := TRUE;
   MM2520_HoldingSidememberInsideLeftInstant.CylinderOperationOld.ToFp := FALSE;
   MM2520_HoldingSidememberInsideLeftInstant.IEC_Timer_0_Instance.PT := T#0MS;
   MM2520_HoldingSidememberInsideLeftInstant.IEC_Timer_0_Instance.IN := FALSE;
   MM2520_HoldingSidememberInsideLeftInstant.R_TRIG_Instance.CLK := FALSE;
   MM2520_HoldingSidememberInsideLeftInstant.R_TRIG_Instance.Q := FALSE;
   MM2520_HoldingSidememberInsideLeftInstant.R_TRIG_Instance.Stat_Bit := FALSE;
   MM2520_HoldingSidememberInsideLeftInstant.IEC_Timer_0_Instance_1.PT := T#0MS;
   MM2520_HoldingSidememberInsideLeftInstant.IEC_Timer_0_Instance_1.IN := FALSE;
   MM2520_HoldingSidememberInsideLeftInstant.IEC_Timer_0_Instance_2.PT := T#0MS;
   MM2520_HoldingSidememberInsideLeftInstant.IEC_Timer_0_Instance_2.IN := FALSE;
   MM2520_HoldingSidememberInsideLeftInstant.IEC_Timer_0_Instance_3.PT := T#0MS;
   MM2520_HoldingSidememberInsideLeftInstant.IEC_Timer_0_Instance_3.IN := FALSE;
   MM2520_HoldingSidememberInsideLeftInstant.IEC_Timer_0_Instance_4.PT := T#0MS;
   MM2520_HoldingSidememberInsideLeftInstant.IEC_Timer_0_Instance_4.IN := TRUE;
   MM2521_HoldingSidememberInsideRightInstant.POWER_OK := TRUE;
   MM2521_HoldingSidememberInsideRightInstant.CylinderNumber := 9;
   MM2521_HoldingSidememberInsideRightInstant.HMICommand := 0;
   MM2521_HoldingSidememberInsideRightInstant.BasicPositionCondition := TRUE;
   MM2521_HoldingSidememberInsideRightInstant.WorkPositionCondition := FALSE;
   MM2521_HoldingSidememberInsideRightInstant.BasicPositionSensor := TRUE;
   MM2521_HoldingSidememberInsideRightInstant.WorkPositionSensor := FALSE;
   MM2521_HoldingSidememberInsideRightInstant.TRIGGER := TRUE;
   MM2521_HoldingSidememberInsideRightInstant.RESET := FALSE;
   MM2521_HoldingSidememberInsideRightInstant.DELAY_BASIC := T#100MS;
   MM2521_HoldingSidememberInsideRightInstant.DELAY_WORK := T#100MS;
   MM2521_HoldingSidememberInsideRightInstant.DELAY_FREE := T#100MS;
   MM2521_HoldingSidememberInsideRightInstant.ERROR_TIME := T#10S;
   MM2521_HoldingSidememberInsideRightInstant.ValveDelay := T#0MS;
   MM2521_HoldingSidememberInsideRightInstant.iNoCollisionBasic := TRUE;
   MM2521_HoldingSidememberInsideRightInstant.iNoCollisionWork := TRUE;
   MM2521_HoldingSidememberInsideRightInstant.iNoCollisionFree := TRUE;
   MM2521_HoldingSidememberInsideRightInstant.VALVE_BASIC := FALSE;
   MM2521_HoldingSidememberInsideRightInstant.VALVE_WORK := FALSE;
   MM2521_HoldingSidememberInsideRightInstant.ERROR_BASIC := FALSE;
   MM2521_HoldingSidememberInsideRightInstant.ERROR_WORK := FALSE;
   MM2521_HoldingSidememberInsideRightInstant.HMIStatus := 1;
   MM2521_HoldingSidememberInsideRightInstant.MOVE_BASIC := FALSE;
   MM2521_HoldingSidememberInsideRightInstant.MOVE_WORK := FALSE;
   MM2521_HoldingSidememberInsideRightInstant.MOVE_FREE := TRUE;
   MM2521_HoldingSidememberInsideRightInstant."4l+Started" := FALSE;
   MM2521_HoldingSidememberInsideRightInstant.InitCommandBP := FALSE;
   MM2521_HoldingSidememberInsideRightInstant.InitCommandWP := FALSE;
   MM2521_HoldingSidememberInsideRightInstant.BasicWorkStartWP := FALSE;
   MM2521_HoldingSidememberInsideRightInstant.BasicWorkStartBP := FALSE;
   MM2521_HoldingSidememberInsideRightInstant.work_valve := FALSE;
   MM2521_HoldingSidememberInsideRightInstant.basic_valve := FALSE;
   MM2521_HoldingSidememberInsideRightInstant.free_valve := FALSE;
   MM2521_HoldingSidememberInsideRightInstant.baspos_error.PT := T#10S;
   MM2521_HoldingSidememberInsideRightInstant.baspos_error.IN := FALSE;
   MM2521_HoldingSidememberInsideRightInstant.workpos_error.PT := T#10S;
   MM2521_HoldingSidememberInsideRightInstant.workpos_error.IN := FALSE;
   MM2521_HoldingSidememberInsideRightInstant.baspos_delay.PT := T#100MS;
   MM2521_HoldingSidememberInsideRightInstant.baspos_delay.IN := FALSE;
   MM2521_HoldingSidememberInsideRightInstant.workpos_delay.PT := T#100MS;
   MM2521_HoldingSidememberInsideRightInstant.workpos_delay.IN := FALSE;
   MM2521_HoldingSidememberInsideRightInstant.CylinderOperationOld.InWp := FALSE;
   MM2521_HoldingSidememberInsideRightInstant.CylinderOperationOld.InBp := TRUE;
   MM2521_HoldingSidememberInsideRightInstant.CylinderOperationOld.InFp := TRUE;
   MM2521_HoldingSidememberInsideRightInstant.CylinderOperationOld.ToWp := FALSE;
   MM2521_HoldingSidememberInsideRightInstant.CylinderOperationOld.ToBp := FALSE;
   MM2521_HoldingSidememberInsideRightInstant.CylinderOperationOld.ToFp := TRUE;
   MM2521_HoldingSidememberInsideRightInstant.IEC_Timer_0_Instance.PT := T#0MS;
   MM2521_HoldingSidememberInsideRightInstant.IEC_Timer_0_Instance.IN := FALSE;
   MM2521_HoldingSidememberInsideRightInstant.R_TRIG_Instance.CLK := FALSE;
   MM2521_HoldingSidememberInsideRightInstant.R_TRIG_Instance.Q := FALSE;
   MM2521_HoldingSidememberInsideRightInstant.R_TRIG_Instance.Stat_Bit := FALSE;
   MM2521_HoldingSidememberInsideRightInstant.IEC_Timer_0_Instance_1.PT := T#0MS;
   MM2521_HoldingSidememberInsideRightInstant.IEC_Timer_0_Instance_1.IN := FALSE;
   MM2521_HoldingSidememberInsideRightInstant.IEC_Timer_0_Instance_2.PT := T#0MS;
   MM2521_HoldingSidememberInsideRightInstant.IEC_Timer_0_Instance_2.IN := FALSE;
   MM2521_HoldingSidememberInsideRightInstant.IEC_Timer_0_Instance_3.PT := T#0MS;
   MM2521_HoldingSidememberInsideRightInstant.IEC_Timer_0_Instance_3.IN := FALSE;
   MM2521_HoldingSidememberInsideRightInstant.IEC_Timer_0_Instance_4.PT := T#0MS;
   MM2521_HoldingSidememberInsideRightInstant.IEC_Timer_0_Instance_4.IN := FALSE;
   MM2540_HoldingSidememberOutsideLeftInstant.POWER_OK := TRUE;
   MM2540_HoldingSidememberOutsideLeftInstant.CylinderNumber := 10;
   MM2540_HoldingSidememberOutsideLeftInstant.HMICommand := 0;
   MM2540_HoldingSidememberOutsideLeftInstant.BasicPositionCondition := TRUE;
   MM2540_HoldingSidememberOutsideLeftInstant.WorkPositionCondition := FALSE;
   MM2540_HoldingSidememberOutsideLeftInstant.BasicPositionSensor := TRUE;
   MM2540_HoldingSidememberOutsideLeftInstant.WorkPositionSensor := FALSE;
   MM2540_HoldingSidememberOutsideLeftInstant.TRIGGER := TRUE;
   MM2540_HoldingSidememberOutsideLeftInstant.RESET := FALSE;
   MM2540_HoldingSidememberOutsideLeftInstant.DELAY_BASIC := T#100MS;
   MM2540_HoldingSidememberOutsideLeftInstant.DELAY_WORK := T#100MS;
   MM2540_HoldingSidememberOutsideLeftInstant.DELAY_FREE := T#100MS;
   MM2540_HoldingSidememberOutsideLeftInstant.ERROR_TIME := T#10S;
   MM2540_HoldingSidememberOutsideLeftInstant.ValveDelay := T#0MS;
   MM2540_HoldingSidememberOutsideLeftInstant.iNoCollisionBasic := TRUE;
   MM2540_HoldingSidememberOutsideLeftInstant.iNoCollisionWork := TRUE;
   MM2540_HoldingSidememberOutsideLeftInstant.iNoCollisionFree := TRUE;
   MM2540_HoldingSidememberOutsideLeftInstant.VALVE_BASIC := FALSE;
   MM2540_HoldingSidememberOutsideLeftInstant.VALVE_WORK := FALSE;
   MM2540_HoldingSidememberOutsideLeftInstant.ERROR_BASIC := FALSE;
   MM2540_HoldingSidememberOutsideLeftInstant.ERROR_WORK := FALSE;
   MM2540_HoldingSidememberOutsideLeftInstant.HMIStatus := 1;
   MM2540_HoldingSidememberOutsideLeftInstant.MOVE_BASIC := FALSE;
   MM2540_HoldingSidememberOutsideLeftInstant.MOVE_WORK := FALSE;
   MM2540_HoldingSidememberOutsideLeftInstant.MOVE_FREE := TRUE;
   MM2540_HoldingSidememberOutsideLeftInstant."4l+Started" := FALSE;
   MM2540_HoldingSidememberOutsideLeftInstant.InitCommandBP := FALSE;
   MM2540_HoldingSidememberOutsideLeftInstant.InitCommandWP := FALSE;
   MM2540_HoldingSidememberOutsideLeftInstant.BasicWorkStartWP := FALSE;
   MM2540_HoldingSidememberOutsideLeftInstant.BasicWorkStartBP := FALSE;
   MM2540_HoldingSidememberOutsideLeftInstant.work_valve := FALSE;
   MM2540_HoldingSidememberOutsideLeftInstant.basic_valve := FALSE;
   MM2540_HoldingSidememberOutsideLeftInstant.free_valve := TRUE;
   MM2540_HoldingSidememberOutsideLeftInstant.baspos_error.PT := T#10S;
   MM2540_HoldingSidememberOutsideLeftInstant.baspos_error.IN := FALSE;
   MM2540_HoldingSidememberOutsideLeftInstant.workpos_error.PT := T#10S;
   MM2540_HoldingSidememberOutsideLeftInstant.workpos_error.IN := FALSE;
   MM2540_HoldingSidememberOutsideLeftInstant.baspos_delay.PT := T#100MS;
   MM2540_HoldingSidememberOutsideLeftInstant.baspos_delay.IN := FALSE;
   MM2540_HoldingSidememberOutsideLeftInstant.workpos_delay.PT := T#100MS;
   MM2540_HoldingSidememberOutsideLeftInstant.workpos_delay.IN := FALSE;
   MM2540_HoldingSidememberOutsideLeftInstant.CylinderOperationOld.InWp := FALSE;
   MM2540_HoldingSidememberOutsideLeftInstant.CylinderOperationOld.InBp := TRUE;
   MM2540_HoldingSidememberOutsideLeftInstant.CylinderOperationOld.InFp := TRUE;
   MM2540_HoldingSidememberOutsideLeftInstant.CylinderOperationOld.ToWp := FALSE;
   MM2540_HoldingSidememberOutsideLeftInstant.CylinderOperationOld.ToBp := FALSE;
   MM2540_HoldingSidememberOutsideLeftInstant.CylinderOperationOld.ToFp := TRUE;
   MM2540_HoldingSidememberOutsideLeftInstant.IEC_Timer_0_Instance.PT := T#0MS;
   MM2540_HoldingSidememberOutsideLeftInstant.IEC_Timer_0_Instance.IN := FALSE;
   MM2540_HoldingSidememberOutsideLeftInstant.R_TRIG_Instance.CLK := FALSE;
   MM2540_HoldingSidememberOutsideLeftInstant.R_TRIG_Instance.Q := FALSE;
   MM2540_HoldingSidememberOutsideLeftInstant.R_TRIG_Instance.Stat_Bit := FALSE;
   MM2540_HoldingSidememberOutsideLeftInstant.IEC_Timer_0_Instance_1.PT := T#0MS;
   MM2540_HoldingSidememberOutsideLeftInstant.IEC_Timer_0_Instance_1.IN := FALSE;
   MM2540_HoldingSidememberOutsideLeftInstant.IEC_Timer_0_Instance_2.PT := T#0MS;
   MM2540_HoldingSidememberOutsideLeftInstant.IEC_Timer_0_Instance_2.IN := FALSE;
   MM2540_HoldingSidememberOutsideLeftInstant.IEC_Timer_0_Instance_3.PT := T#0MS;
   MM2540_HoldingSidememberOutsideLeftInstant.IEC_Timer_0_Instance_3.IN := FALSE;
   MM2540_HoldingSidememberOutsideLeftInstant.IEC_Timer_0_Instance_4.PT := T#0MS;
   MM2540_HoldingSidememberOutsideLeftInstant.IEC_Timer_0_Instance_4.IN := FALSE;
   MM2541_HoldingSidememberOutsideRightInstant.POWER_OK := TRUE;
   MM2541_HoldingSidememberOutsideRightInstant.CylinderNumber := 11;
   MM2541_HoldingSidememberOutsideRightInstant.HMICommand := 0;
   MM2541_HoldingSidememberOutsideRightInstant.BasicPositionCondition := TRUE;
   MM2541_HoldingSidememberOutsideRightInstant.WorkPositionCondition := FALSE;
   MM2541_HoldingSidememberOutsideRightInstant.BasicPositionSensor := TRUE;
   MM2541_HoldingSidememberOutsideRightInstant.WorkPositionSensor := FALSE;
   MM2541_HoldingSidememberOutsideRightInstant.TRIGGER := TRUE;
   MM2541_HoldingSidememberOutsideRightInstant.RESET := FALSE;
   MM2541_HoldingSidememberOutsideRightInstant.DELAY_BASIC := T#100MS;
   MM2541_HoldingSidememberOutsideRightInstant.DELAY_WORK := T#100MS;
   MM2541_HoldingSidememberOutsideRightInstant.DELAY_FREE := T#100MS;
   MM2541_HoldingSidememberOutsideRightInstant.ERROR_TIME := T#10S;
   MM2541_HoldingSidememberOutsideRightInstant.ValveDelay := T#0MS;
   MM2541_HoldingSidememberOutsideRightInstant.iNoCollisionBasic := TRUE;
   MM2541_HoldingSidememberOutsideRightInstant.iNoCollisionWork := TRUE;
   MM2541_HoldingSidememberOutsideRightInstant.iNoCollisionFree := TRUE;
   MM2541_HoldingSidememberOutsideRightInstant.VALVE_BASIC := TRUE;
   MM2541_HoldingSidememberOutsideRightInstant.VALVE_WORK := FALSE;
   MM2541_HoldingSidememberOutsideRightInstant.ERROR_BASIC := FALSE;
   MM2541_HoldingSidememberOutsideRightInstant.ERROR_WORK := FALSE;
   MM2541_HoldingSidememberOutsideRightInstant.HMIStatus := 257;
   MM2541_HoldingSidememberOutsideRightInstant.MOVE_BASIC := TRUE;
   MM2541_HoldingSidememberOutsideRightInstant.MOVE_WORK := FALSE;
   MM2541_HoldingSidememberOutsideRightInstant.MOVE_FREE := FALSE;
   MM2541_HoldingSidememberOutsideRightInstant."4l+Started" := FALSE;
   MM2541_HoldingSidememberOutsideRightInstant.InitCommandBP := FALSE;
   MM2541_HoldingSidememberOutsideRightInstant.InitCommandWP := FALSE;
   MM2541_HoldingSidememberOutsideRightInstant.BasicWorkStartWP := FALSE;
   MM2541_HoldingSidememberOutsideRightInstant.BasicWorkStartBP := FALSE;
   MM2541_HoldingSidememberOutsideRightInstant.work_valve := FALSE;
   MM2541_HoldingSidememberOutsideRightInstant.basic_valve := TRUE;
   MM2541_HoldingSidememberOutsideRightInstant.free_valve := TRUE;
   MM2541_HoldingSidememberOutsideRightInstant.baspos_error.PT := T#10S;
   MM2541_HoldingSidememberOutsideRightInstant.baspos_error.IN := FALSE;
   MM2541_HoldingSidememberOutsideRightInstant.workpos_error.PT := T#10S;
   MM2541_HoldingSidememberOutsideRightInstant.workpos_error.IN := FALSE;
   MM2541_HoldingSidememberOutsideRightInstant.baspos_delay.PT := T#100MS;
   MM2541_HoldingSidememberOutsideRightInstant.baspos_delay.IN := TRUE;
   MM2541_HoldingSidememberOutsideRightInstant.workpos_delay.PT := T#100MS;
   MM2541_HoldingSidememberOutsideRightInstant.workpos_delay.IN := FALSE;
   MM2541_HoldingSidememberOutsideRightInstant.CylinderOperationOld.InWp := FALSE;
   MM2541_HoldingSidememberOutsideRightInstant.CylinderOperationOld.InBp := TRUE;
   MM2541_HoldingSidememberOutsideRightInstant.CylinderOperationOld.InFp := FALSE;
   MM2541_HoldingSidememberOutsideRightInstant.CylinderOperationOld.ToWp := FALSE;
   MM2541_HoldingSidememberOutsideRightInstant.CylinderOperationOld.ToBp := TRUE;
   MM2541_HoldingSidememberOutsideRightInstant.CylinderOperationOld.ToFp := FALSE;
   MM2541_HoldingSidememberOutsideRightInstant.IEC_Timer_0_Instance.PT := T#0MS;
   MM2541_HoldingSidememberOutsideRightInstant.IEC_Timer_0_Instance.IN := FALSE;
   MM2541_HoldingSidememberOutsideRightInstant.R_TRIG_Instance.CLK := FALSE;
   MM2541_HoldingSidememberOutsideRightInstant.R_TRIG_Instance.Q := FALSE;
   MM2541_HoldingSidememberOutsideRightInstant.R_TRIG_Instance.Stat_Bit := FALSE;
   MM2541_HoldingSidememberOutsideRightInstant.IEC_Timer_0_Instance_1.PT := T#0MS;
   MM2541_HoldingSidememberOutsideRightInstant.IEC_Timer_0_Instance_1.IN := FALSE;
   MM2541_HoldingSidememberOutsideRightInstant.IEC_Timer_0_Instance_2.PT := T#0MS;
   MM2541_HoldingSidememberOutsideRightInstant.IEC_Timer_0_Instance_2.IN := FALSE;
   MM2541_HoldingSidememberOutsideRightInstant.IEC_Timer_0_Instance_3.PT := T#0MS;
   MM2541_HoldingSidememberOutsideRightInstant.IEC_Timer_0_Instance_3.IN := FALSE;
   MM2541_HoldingSidememberOutsideRightInstant.IEC_Timer_0_Instance_4.PT := T#0MS;
   MM2541_HoldingSidememberOutsideRightInstant.IEC_Timer_0_Instance_4.IN := TRUE;
   MM300_ShiftingSupportRightInstant.POWER_OK := TRUE;
   MM300_ShiftingSupportRightInstant.CylinderNumber := 12;
   MM300_ShiftingSupportRightInstant.HMICommand := 0;
   MM300_ShiftingSupportRightInstant.BasicPositionCondition := TRUE;
   MM300_ShiftingSupportRightInstant.WorkPositionCondition := FALSE;
   MM300_ShiftingSupportRightInstant.BasicPositionSensor := TRUE;
   MM300_ShiftingSupportRightInstant.WorkPositionSensor := FALSE;
   MM300_ShiftingSupportRightInstant.TRIGGER := TRUE;
   MM300_ShiftingSupportRightInstant.RESET := FALSE;
   MM300_ShiftingSupportRightInstant.DELAY_BASIC := T#100MS;
   MM300_ShiftingSupportRightInstant.DELAY_WORK := T#100MS;
   MM300_ShiftingSupportRightInstant.DELAY_FREE := T#100MS;
   MM300_ShiftingSupportRightInstant.ERROR_TIME := T#10S;
   MM300_ShiftingSupportRightInstant.ValveDelay := T#0MS;
   MM300_ShiftingSupportRightInstant.iNoCollisionBasic := TRUE;
   MM300_ShiftingSupportRightInstant.iNoCollisionWork := TRUE;
   MM300_ShiftingSupportRightInstant.iNoCollisionFree := TRUE;
   MM300_ShiftingSupportRightInstant.VALVE_BASIC := TRUE;
   MM300_ShiftingSupportRightInstant.VALVE_WORK := FALSE;
   MM300_ShiftingSupportRightInstant.ERROR_BASIC := FALSE;
   MM300_ShiftingSupportRightInstant.ERROR_WORK := FALSE;
   MM300_ShiftingSupportRightInstant.HMIStatus := 257;
   MM300_ShiftingSupportRightInstant.MOVE_BASIC := TRUE;
   MM300_ShiftingSupportRightInstant.MOVE_WORK := FALSE;
   MM300_ShiftingSupportRightInstant.MOVE_FREE := FALSE;
   MM300_ShiftingSupportRightInstant."4l+Started" := FALSE;
   MM300_ShiftingSupportRightInstant.InitCommandBP := FALSE;
   MM300_ShiftingSupportRightInstant.InitCommandWP := FALSE;
   MM300_ShiftingSupportRightInstant.BasicWorkStartWP := FALSE;
   MM300_ShiftingSupportRightInstant.BasicWorkStartBP := FALSE;
   MM300_ShiftingSupportRightInstant.work_valve := FALSE;
   MM300_ShiftingSupportRightInstant.basic_valve := TRUE;
   MM300_ShiftingSupportRightInstant.free_valve := TRUE;
   MM300_ShiftingSupportRightInstant.baspos_error.PT := T#10S;
   MM300_ShiftingSupportRightInstant.baspos_error.IN := FALSE;
   MM300_ShiftingSupportRightInstant.workpos_error.PT := T#10S;
   MM300_ShiftingSupportRightInstant.workpos_error.IN := FALSE;
   MM300_ShiftingSupportRightInstant.baspos_delay.PT := T#100MS;
   MM300_ShiftingSupportRightInstant.baspos_delay.IN := TRUE;
   MM300_ShiftingSupportRightInstant.workpos_delay.PT := T#100MS;
   MM300_ShiftingSupportRightInstant.workpos_delay.IN := FALSE;
   MM300_ShiftingSupportRightInstant.CylinderOperationOld.InWp := FALSE;
   MM300_ShiftingSupportRightInstant.CylinderOperationOld.InBp := TRUE;
   MM300_ShiftingSupportRightInstant.CylinderOperationOld.InFp := FALSE;
   MM300_ShiftingSupportRightInstant.CylinderOperationOld.ToWp := FALSE;
   MM300_ShiftingSupportRightInstant.CylinderOperationOld.ToBp := TRUE;
   MM300_ShiftingSupportRightInstant.CylinderOperationOld.ToFp := FALSE;
   MM300_ShiftingSupportRightInstant.IEC_Timer_0_Instance.PT := T#0MS;
   MM300_ShiftingSupportRightInstant.IEC_Timer_0_Instance.IN := FALSE;
   MM300_ShiftingSupportRightInstant.R_TRIG_Instance.CLK := FALSE;
   MM300_ShiftingSupportRightInstant.R_TRIG_Instance.Q := FALSE;
   MM300_ShiftingSupportRightInstant.R_TRIG_Instance.Stat_Bit := FALSE;
   MM300_ShiftingSupportRightInstant.IEC_Timer_0_Instance_1.PT := T#0MS;
   MM300_ShiftingSupportRightInstant.IEC_Timer_0_Instance_1.IN := FALSE;
   MM300_ShiftingSupportRightInstant.IEC_Timer_0_Instance_2.PT := T#0MS;
   MM300_ShiftingSupportRightInstant.IEC_Timer_0_Instance_2.IN := FALSE;
   MM300_ShiftingSupportRightInstant.IEC_Timer_0_Instance_3.PT := T#0MS;
   MM300_ShiftingSupportRightInstant.IEC_Timer_0_Instance_3.IN := FALSE;
   MM300_ShiftingSupportRightInstant.IEC_Timer_0_Instance_4.PT := T#0MS;
   MM300_ShiftingSupportRightInstant.IEC_Timer_0_Instance_4.IN := TRUE;
   MM302_ShiftingSupportLeftInstant.POWER_OK := TRUE;
   MM302_ShiftingSupportLeftInstant.CylinderNumber := 13;
   MM302_ShiftingSupportLeftInstant.HMICommand := 0;
   MM302_ShiftingSupportLeftInstant.BasicPositionCondition := TRUE;
   MM302_ShiftingSupportLeftInstant.WorkPositionCondition := FALSE;
   MM302_ShiftingSupportLeftInstant.BasicPositionSensor := TRUE;
   MM302_ShiftingSupportLeftInstant.WorkPositionSensor := FALSE;
   MM302_ShiftingSupportLeftInstant.TRIGGER := TRUE;
   MM302_ShiftingSupportLeftInstant.RESET := FALSE;
   MM302_ShiftingSupportLeftInstant.DELAY_BASIC := T#100MS;
   MM302_ShiftingSupportLeftInstant.DELAY_WORK := T#100MS;
   MM302_ShiftingSupportLeftInstant.DELAY_FREE := T#100MS;
   MM302_ShiftingSupportLeftInstant.ERROR_TIME := T#10S;
   MM302_ShiftingSupportLeftInstant.ValveDelay := T#0MS;
   MM302_ShiftingSupportLeftInstant.iNoCollisionBasic := TRUE;
   MM302_ShiftingSupportLeftInstant.iNoCollisionWork := TRUE;
   MM302_ShiftingSupportLeftInstant.iNoCollisionFree := TRUE;
   MM302_ShiftingSupportLeftInstant.VALVE_BASIC := TRUE;
   MM302_ShiftingSupportLeftInstant.VALVE_WORK := FALSE;
   MM302_ShiftingSupportLeftInstant.ERROR_BASIC := FALSE;
   MM302_ShiftingSupportLeftInstant.ERROR_WORK := FALSE;
   MM302_ShiftingSupportLeftInstant.HMIStatus := 257;
   MM302_ShiftingSupportLeftInstant.MOVE_BASIC := TRUE;
   MM302_ShiftingSupportLeftInstant.MOVE_WORK := FALSE;
   MM302_ShiftingSupportLeftInstant.MOVE_FREE := FALSE;
   MM302_ShiftingSupportLeftInstant."4l+Started" := FALSE;
   MM302_ShiftingSupportLeftInstant.InitCommandBP := FALSE;
   MM302_ShiftingSupportLeftInstant.InitCommandWP := FALSE;
   MM302_ShiftingSupportLeftInstant.BasicWorkStartWP := FALSE;
   MM302_ShiftingSupportLeftInstant.BasicWorkStartBP := FALSE;
   MM302_ShiftingSupportLeftInstant.work_valve := FALSE;
   MM302_ShiftingSupportLeftInstant.basic_valve := TRUE;
   MM302_ShiftingSupportLeftInstant.free_valve := TRUE;
   MM302_ShiftingSupportLeftInstant.baspos_error.PT := T#10S;
   MM302_ShiftingSupportLeftInstant.baspos_error.IN := FALSE;
   MM302_ShiftingSupportLeftInstant.workpos_error.PT := T#10S;
   MM302_ShiftingSupportLeftInstant.workpos_error.IN := FALSE;
   MM302_ShiftingSupportLeftInstant.baspos_delay.PT := T#100MS;
   MM302_ShiftingSupportLeftInstant.baspos_delay.IN := TRUE;
   MM302_ShiftingSupportLeftInstant.workpos_delay.PT := T#100MS;
   MM302_ShiftingSupportLeftInstant.workpos_delay.IN := FALSE;
   MM302_ShiftingSupportLeftInstant.CylinderOperationOld.InWp := FALSE;
   MM302_ShiftingSupportLeftInstant.CylinderOperationOld.InBp := TRUE;
   MM302_ShiftingSupportLeftInstant.CylinderOperationOld.InFp := FALSE;
   MM302_ShiftingSupportLeftInstant.CylinderOperationOld.ToWp := FALSE;
   MM302_ShiftingSupportLeftInstant.CylinderOperationOld.ToBp := TRUE;
   MM302_ShiftingSupportLeftInstant.CylinderOperationOld.ToFp := FALSE;
   MM302_ShiftingSupportLeftInstant.IEC_Timer_0_Instance.PT := T#0MS;
   MM302_ShiftingSupportLeftInstant.IEC_Timer_0_Instance.IN := FALSE;
   MM302_ShiftingSupportLeftInstant.R_TRIG_Instance.CLK := FALSE;
   MM302_ShiftingSupportLeftInstant.R_TRIG_Instance.Q := FALSE;
   MM302_ShiftingSupportLeftInstant.R_TRIG_Instance.Stat_Bit := FALSE;
   MM302_ShiftingSupportLeftInstant.IEC_Timer_0_Instance_1.PT := T#0MS;
   MM302_ShiftingSupportLeftInstant.IEC_Timer_0_Instance_1.IN := FALSE;
   MM302_ShiftingSupportLeftInstant.IEC_Timer_0_Instance_2.PT := T#0MS;
   MM302_ShiftingSupportLeftInstant.IEC_Timer_0_Instance_2.IN := FALSE;
   MM302_ShiftingSupportLeftInstant.IEC_Timer_0_Instance_3.PT := T#0MS;
   MM302_ShiftingSupportLeftInstant.IEC_Timer_0_Instance_3.IN := FALSE;
   MM302_ShiftingSupportLeftInstant.IEC_Timer_0_Instance_4.PT := T#0MS;
   MM302_ShiftingSupportLeftInstant.IEC_Timer_0_Instance_4.IN := TRUE;
   MM304_MovingStopRightInstant.POWER_OK := TRUE;
   MM304_MovingStopRightInstant.CylinderNumber := 14;
   MM304_MovingStopRightInstant.HMICommand := 0;
   MM304_MovingStopRightInstant.BasicPositionCondition := TRUE;
   MM304_MovingStopRightInstant.WorkPositionCondition := FALSE;
   MM304_MovingStopRightInstant.BasicPositionSensor := TRUE;
   MM304_MovingStopRightInstant.WorkPositionSensor := FALSE;
   MM304_MovingStopRightInstant.TRIGGER := TRUE;
   MM304_MovingStopRightInstant.RESET := FALSE;
   MM304_MovingStopRightInstant.DELAY_BASIC := T#100MS;
   MM304_MovingStopRightInstant.DELAY_WORK := T#100MS;
   MM304_MovingStopRightInstant.DELAY_FREE := T#100MS;
   MM304_MovingStopRightInstant.ERROR_TIME := T#10S;
   MM304_MovingStopRightInstant.ValveDelay := T#0MS;
   MM304_MovingStopRightInstant.iNoCollisionBasic := TRUE;
   MM304_MovingStopRightInstant.iNoCollisionWork := TRUE;
   MM304_MovingStopRightInstant.iNoCollisionFree := TRUE;
   MM304_MovingStopRightInstant.VALVE_BASIC := TRUE;
   MM304_MovingStopRightInstant.VALVE_WORK := FALSE;
   MM304_MovingStopRightInstant.ERROR_BASIC := FALSE;
   MM304_MovingStopRightInstant.ERROR_WORK := FALSE;
   MM304_MovingStopRightInstant.HMIStatus := 257;
   MM304_MovingStopRightInstant.MOVE_BASIC := TRUE;
   MM304_MovingStopRightInstant.MOVE_WORK := FALSE;
   MM304_MovingStopRightInstant.MOVE_FREE := FALSE;
   MM304_MovingStopRightInstant."4l+Started" := FALSE;
   MM304_MovingStopRightInstant.InitCommandBP := FALSE;
   MM304_MovingStopRightInstant.InitCommandWP := FALSE;
   MM304_MovingStopRightInstant.BasicWorkStartWP := FALSE;
   MM304_MovingStopRightInstant.BasicWorkStartBP := FALSE;
   MM304_MovingStopRightInstant.work_valve := FALSE;
   MM304_MovingStopRightInstant.basic_valve := TRUE;
   MM304_MovingStopRightInstant.free_valve := TRUE;
   MM304_MovingStopRightInstant.baspos_error.PT := T#10S;
   MM304_MovingStopRightInstant.baspos_error.IN := FALSE;
   MM304_MovingStopRightInstant.workpos_error.PT := T#10S;
   MM304_MovingStopRightInstant.workpos_error.IN := FALSE;
   MM304_MovingStopRightInstant.baspos_delay.PT := T#100MS;
   MM304_MovingStopRightInstant.baspos_delay.IN := TRUE;
   MM304_MovingStopRightInstant.workpos_delay.PT := T#100MS;
   MM304_MovingStopRightInstant.workpos_delay.IN := FALSE;
   MM304_MovingStopRightInstant.CylinderOperationOld.InWp := FALSE;
   MM304_MovingStopRightInstant.CylinderOperationOld.InBp := TRUE;
   MM304_MovingStopRightInstant.CylinderOperationOld.InFp := FALSE;
   MM304_MovingStopRightInstant.CylinderOperationOld.ToWp := FALSE;
   MM304_MovingStopRightInstant.CylinderOperationOld.ToBp := TRUE;
   MM304_MovingStopRightInstant.CylinderOperationOld.ToFp := FALSE;
   MM304_MovingStopRightInstant.IEC_Timer_0_Instance.PT := T#0MS;
   MM304_MovingStopRightInstant.IEC_Timer_0_Instance.IN := FALSE;
   MM304_MovingStopRightInstant.R_TRIG_Instance.CLK := FALSE;
   MM304_MovingStopRightInstant.R_TRIG_Instance.Q := FALSE;
   MM304_MovingStopRightInstant.R_TRIG_Instance.Stat_Bit := FALSE;
   MM304_MovingStopRightInstant.IEC_Timer_0_Instance_1.PT := T#0MS;
   MM304_MovingStopRightInstant.IEC_Timer_0_Instance_1.IN := FALSE;
   MM304_MovingStopRightInstant.IEC_Timer_0_Instance_2.PT := T#0MS;
   MM304_MovingStopRightInstant.IEC_Timer_0_Instance_2.IN := FALSE;
   MM304_MovingStopRightInstant.IEC_Timer_0_Instance_3.PT := T#0MS;
   MM304_MovingStopRightInstant.IEC_Timer_0_Instance_3.IN := FALSE;
   MM304_MovingStopRightInstant.IEC_Timer_0_Instance_4.PT := T#0MS;
   MM304_MovingStopRightInstant.IEC_Timer_0_Instance_4.IN := TRUE;
   MM306_MovingStopLeftInstant.POWER_OK := TRUE;
   MM306_MovingStopLeftInstant.CylinderNumber := 15;
   MM306_MovingStopLeftInstant.HMICommand := 0;
   MM306_MovingStopLeftInstant.BasicPositionCondition := TRUE;
   MM306_MovingStopLeftInstant.WorkPositionCondition := FALSE;
   MM306_MovingStopLeftInstant.BasicPositionSensor := TRUE;
   MM306_MovingStopLeftInstant.WorkPositionSensor := FALSE;
   MM306_MovingStopLeftInstant.TRIGGER := TRUE;
   MM306_MovingStopLeftInstant.RESET := FALSE;
   MM306_MovingStopLeftInstant.DELAY_BASIC := T#100MS;
   MM306_MovingStopLeftInstant.DELAY_WORK := T#100MS;
   MM306_MovingStopLeftInstant.DELAY_FREE := T#100MS;
   MM306_MovingStopLeftInstant.ERROR_TIME := T#10S;
   MM306_MovingStopLeftInstant.ValveDelay := T#0MS;
   MM306_MovingStopLeftInstant.iNoCollisionBasic := TRUE;
   MM306_MovingStopLeftInstant.iNoCollisionWork := TRUE;
   MM306_MovingStopLeftInstant.iNoCollisionFree := TRUE;
   MM306_MovingStopLeftInstant.VALVE_BASIC := FALSE;
   MM306_MovingStopLeftInstant.VALVE_WORK := FALSE;
   MM306_MovingStopLeftInstant.ERROR_BASIC := FALSE;
   MM306_MovingStopLeftInstant.ERROR_WORK := FALSE;
   MM306_MovingStopLeftInstant.HMIStatus := 1;
   MM306_MovingStopLeftInstant.MOVE_BASIC := FALSE;
   MM306_MovingStopLeftInstant.MOVE_WORK := FALSE;
   MM306_MovingStopLeftInstant.MOVE_FREE := TRUE;
   MM306_MovingStopLeftInstant."4l+Started" := FALSE;
   MM306_MovingStopLeftInstant.InitCommandBP := FALSE;
   MM306_MovingStopLeftInstant.InitCommandWP := FALSE;
   MM306_MovingStopLeftInstant.BasicWorkStartWP := FALSE;
   MM306_MovingStopLeftInstant.BasicWorkStartBP := FALSE;
   MM306_MovingStopLeftInstant.work_valve := FALSE;
   MM306_MovingStopLeftInstant.basic_valve := FALSE;
   MM306_MovingStopLeftInstant.free_valve := FALSE;
   MM306_MovingStopLeftInstant.baspos_error.PT := T#0MS;
   MM306_MovingStopLeftInstant.baspos_error.IN := FALSE;
   MM306_MovingStopLeftInstant.workpos_error.PT := T#0MS;
   MM306_MovingStopLeftInstant.workpos_error.IN := FALSE;
   MM306_MovingStopLeftInstant.baspos_delay.PT := T#0MS;
   MM306_MovingStopLeftInstant.baspos_delay.IN := FALSE;
   MM306_MovingStopLeftInstant.workpos_delay.PT := T#0MS;
   MM306_MovingStopLeftInstant.workpos_delay.IN := FALSE;
   MM306_MovingStopLeftInstant.CylinderOperationOld.InWp := FALSE;
   MM306_MovingStopLeftInstant.CylinderOperationOld.InBp := TRUE;
   MM306_MovingStopLeftInstant.CylinderOperationOld.InFp := TRUE;
   MM306_MovingStopLeftInstant.CylinderOperationOld.ToWp := FALSE;
   MM306_MovingStopLeftInstant.CylinderOperationOld.ToBp := FALSE;
   MM306_MovingStopLeftInstant.CylinderOperationOld.ToFp := TRUE;
   MM306_MovingStopLeftInstant.IEC_Timer_0_Instance.PT := T#0MS;
   MM306_MovingStopLeftInstant.IEC_Timer_0_Instance.IN := FALSE;
   MM306_MovingStopLeftInstant.R_TRIG_Instance.CLK := FALSE;
   MM306_MovingStopLeftInstant.R_TRIG_Instance.Q := FALSE;
   MM306_MovingStopLeftInstant.R_TRIG_Instance.Stat_Bit := FALSE;
   MM306_MovingStopLeftInstant.IEC_Timer_0_Instance_1.PT := T#0MS;
   MM306_MovingStopLeftInstant.IEC_Timer_0_Instance_1.IN := FALSE;
   MM306_MovingStopLeftInstant.IEC_Timer_0_Instance_2.PT := T#0MS;
   MM306_MovingStopLeftInstant.IEC_Timer_0_Instance_2.IN := FALSE;
   MM306_MovingStopLeftInstant.IEC_Timer_0_Instance_3.PT := T#0MS;
   MM306_MovingStopLeftInstant.IEC_Timer_0_Instance_3.IN := FALSE;
   MM306_MovingStopLeftInstant.IEC_Timer_0_Instance_4.PT := T#0MS;
   MM306_MovingStopLeftInstant.IEC_Timer_0_Instance_4.IN := FALSE;
   MM340_RivetingUnitRightInstant.POWER_OK := TRUE;
   MM340_RivetingUnitRightInstant.CylinderNumber := 16;
   MM340_RivetingUnitRightInstant.HMICommand := 0;
   MM340_RivetingUnitRightInstant.BasicPositionCondition := TRUE;
   MM340_RivetingUnitRightInstant.WorkPositionCondition := FALSE;
   MM340_RivetingUnitRightInstant.BasicPositionSensor := TRUE;
   MM340_RivetingUnitRightInstant.WorkPositionSensor := FALSE;
   MM340_RivetingUnitRightInstant.TRIGGER := TRUE;
   MM340_RivetingUnitRightInstant.RESET := FALSE;
   MM340_RivetingUnitRightInstant.DELAY_BASIC := T#100MS;
   MM340_RivetingUnitRightInstant.DELAY_WORK := T#100MS;
   MM340_RivetingUnitRightInstant.DELAY_FREE := T#100MS;
   MM340_RivetingUnitRightInstant.ERROR_TIME := T#10S;
   MM340_RivetingUnitRightInstant.ValveDelay := T#0MS;
   MM340_RivetingUnitRightInstant.iNoCollisionBasic := TRUE;
   MM340_RivetingUnitRightInstant.iNoCollisionWork := TRUE;
   MM340_RivetingUnitRightInstant.iNoCollisionFree := TRUE;
   MM340_RivetingUnitRightInstant.VALVE_BASIC := FALSE;
   MM340_RivetingUnitRightInstant.VALVE_WORK := FALSE;
   MM340_RivetingUnitRightInstant.ERROR_BASIC := FALSE;
   MM340_RivetingUnitRightInstant.ERROR_WORK := FALSE;
   MM340_RivetingUnitRightInstant.HMIStatus := 1;
   MM340_RivetingUnitRightInstant.MOVE_BASIC := FALSE;
   MM340_RivetingUnitRightInstant.MOVE_WORK := FALSE;
   MM340_RivetingUnitRightInstant.MOVE_FREE := TRUE;
   MM340_RivetingUnitRightInstant."4l+Started" := FALSE;
   MM340_RivetingUnitRightInstant.InitCommandBP := FALSE;
   MM340_RivetingUnitRightInstant.InitCommandWP := FALSE;
   MM340_RivetingUnitRightInstant.BasicWorkStartWP := FALSE;
   MM340_RivetingUnitRightInstant.BasicWorkStartBP := FALSE;
   MM340_RivetingUnitRightInstant.work_valve := FALSE;
   MM340_RivetingUnitRightInstant.basic_valve := FALSE;
   MM340_RivetingUnitRightInstant.free_valve := FALSE;
   MM340_RivetingUnitRightInstant.baspos_error.PT := T#0MS;
   MM340_RivetingUnitRightInstant.baspos_error.IN := FALSE;
   MM340_RivetingUnitRightInstant.workpos_error.PT := T#0MS;
   MM340_RivetingUnitRightInstant.workpos_error.IN := FALSE;
   MM340_RivetingUnitRightInstant.baspos_delay.PT := T#0MS;
   MM340_RivetingUnitRightInstant.baspos_delay.IN := FALSE;
   MM340_RivetingUnitRightInstant.workpos_delay.PT := T#0MS;
   MM340_RivetingUnitRightInstant.workpos_delay.IN := FALSE;
   MM340_RivetingUnitRightInstant.CylinderOperationOld.InWp := FALSE;
   MM340_RivetingUnitRightInstant.CylinderOperationOld.InBp := TRUE;
   MM340_RivetingUnitRightInstant.CylinderOperationOld.InFp := TRUE;
   MM340_RivetingUnitRightInstant.CylinderOperationOld.ToWp := FALSE;
   MM340_RivetingUnitRightInstant.CylinderOperationOld.ToBp := FALSE;
   MM340_RivetingUnitRightInstant.CylinderOperationOld.ToFp := TRUE;
   MM340_RivetingUnitRightInstant.IEC_Timer_0_Instance.PT := T#0MS;
   MM340_RivetingUnitRightInstant.IEC_Timer_0_Instance.IN := FALSE;
   MM340_RivetingUnitRightInstant.R_TRIG_Instance.CLK := FALSE;
   MM340_RivetingUnitRightInstant.R_TRIG_Instance.Q := FALSE;
   MM340_RivetingUnitRightInstant.R_TRIG_Instance.Stat_Bit := FALSE;
   MM340_RivetingUnitRightInstant.IEC_Timer_0_Instance_1.PT := T#0MS;
   MM340_RivetingUnitRightInstant.IEC_Timer_0_Instance_1.IN := FALSE;
   MM340_RivetingUnitRightInstant.IEC_Timer_0_Instance_2.PT := T#0MS;
   MM340_RivetingUnitRightInstant.IEC_Timer_0_Instance_2.IN := FALSE;
   MM340_RivetingUnitRightInstant.IEC_Timer_0_Instance_3.PT := T#0MS;
   MM340_RivetingUnitRightInstant.IEC_Timer_0_Instance_3.IN := FALSE;
   MM340_RivetingUnitRightInstant.IEC_Timer_0_Instance_4.PT := T#0MS;
   MM340_RivetingUnitRightInstant.IEC_Timer_0_Instance_4.IN := FALSE;
   MM342_RivetingUnitLeftInstant.POWER_OK := TRUE;
   MM342_RivetingUnitLeftInstant.CylinderNumber := 17;
   MM342_RivetingUnitLeftInstant.HMICommand := 0;
   MM342_RivetingUnitLeftInstant.BasicPositionCondition := FALSE;
   MM342_RivetingUnitLeftInstant.WorkPositionCondition := TRUE;
   MM342_RivetingUnitLeftInstant.BasicPositionSensor := FALSE;
   MM342_RivetingUnitLeftInstant.WorkPositionSensor := TRUE;
   MM342_RivetingUnitLeftInstant.TRIGGER := TRUE;
   MM342_RivetingUnitLeftInstant.RESET := FALSE;
   MM342_RivetingUnitLeftInstant.DELAY_BASIC := T#100MS;
   MM342_RivetingUnitLeftInstant.DELAY_WORK := T#100MS;
   MM342_RivetingUnitLeftInstant.DELAY_FREE := T#100MS;
   MM342_RivetingUnitLeftInstant.ERROR_TIME := T#10S;
   MM342_RivetingUnitLeftInstant.ValveDelay := T#0MS;
   MM342_RivetingUnitLeftInstant.iNoCollisionBasic := TRUE;
   MM342_RivetingUnitLeftInstant.iNoCollisionWork := TRUE;
   MM342_RivetingUnitLeftInstant.iNoCollisionFree := TRUE;
   MM342_RivetingUnitLeftInstant.VALVE_BASIC := FALSE;
   MM342_RivetingUnitLeftInstant.VALVE_WORK := FALSE;
   MM342_RivetingUnitLeftInstant.ERROR_BASIC := FALSE;
   MM342_RivetingUnitLeftInstant.ERROR_WORK := FALSE;
   MM342_RivetingUnitLeftInstant.HMIStatus := 2;
   MM342_RivetingUnitLeftInstant.MOVE_BASIC := FALSE;
   MM342_RivetingUnitLeftInstant.MOVE_WORK := FALSE;
   MM342_RivetingUnitLeftInstant.MOVE_FREE := TRUE;
   MM342_RivetingUnitLeftInstant."4l+Started" := FALSE;
   MM342_RivetingUnitLeftInstant.InitCommandBP := FALSE;
   MM342_RivetingUnitLeftInstant.InitCommandWP := FALSE;
   MM342_RivetingUnitLeftInstant.BasicWorkStartWP := FALSE;
   MM342_RivetingUnitLeftInstant.BasicWorkStartBP := FALSE;
   MM342_RivetingUnitLeftInstant.work_valve := FALSE;
   MM342_RivetingUnitLeftInstant.basic_valve := FALSE;
   MM342_RivetingUnitLeftInstant.free_valve := FALSE;
   MM342_RivetingUnitLeftInstant.baspos_error.PT := T#0MS;
   MM342_RivetingUnitLeftInstant.baspos_error.IN := FALSE;
   MM342_RivetingUnitLeftInstant.workpos_error.PT := T#0MS;
   MM342_RivetingUnitLeftInstant.workpos_error.IN := FALSE;
   MM342_RivetingUnitLeftInstant.baspos_delay.PT := T#0MS;
   MM342_RivetingUnitLeftInstant.baspos_delay.IN := FALSE;
   MM342_RivetingUnitLeftInstant.workpos_delay.PT := T#0MS;
   MM342_RivetingUnitLeftInstant.workpos_delay.IN := FALSE;
   MM342_RivetingUnitLeftInstant.CylinderOperationOld.InWp := TRUE;
   MM342_RivetingUnitLeftInstant.CylinderOperationOld.InBp := FALSE;
   MM342_RivetingUnitLeftInstant.CylinderOperationOld.InFp := TRUE;
   MM342_RivetingUnitLeftInstant.CylinderOperationOld.ToWp := FALSE;
   MM342_RivetingUnitLeftInstant.CylinderOperationOld.ToBp := FALSE;
   MM342_RivetingUnitLeftInstant.CylinderOperationOld.ToFp := TRUE;
   MM342_RivetingUnitLeftInstant.IEC_Timer_0_Instance.PT := T#0MS;
   MM342_RivetingUnitLeftInstant.IEC_Timer_0_Instance.IN := FALSE;
   MM342_RivetingUnitLeftInstant.R_TRIG_Instance.CLK := FALSE;
   MM342_RivetingUnitLeftInstant.R_TRIG_Instance.Q := FALSE;
   MM342_RivetingUnitLeftInstant.R_TRIG_Instance.Stat_Bit := FALSE;
   MM342_RivetingUnitLeftInstant.IEC_Timer_0_Instance_1.PT := T#0MS;
   MM342_RivetingUnitLeftInstant.IEC_Timer_0_Instance_1.IN := FALSE;
   MM342_RivetingUnitLeftInstant.IEC_Timer_0_Instance_2.PT := T#0MS;
   MM342_RivetingUnitLeftInstant.IEC_Timer_0_Instance_2.IN := FALSE;
   MM342_RivetingUnitLeftInstant.IEC_Timer_0_Instance_3.PT := T#0MS;
   MM342_RivetingUnitLeftInstant.IEC_Timer_0_Instance_3.IN := FALSE;
   MM342_RivetingUnitLeftInstant.IEC_Timer_0_Instance_4.PT := T#0MS;
   MM342_RivetingUnitLeftInstant.IEC_Timer_0_Instance_4.IN := FALSE;
   MM344_RivetingSupportRightInstant.POWER_OK := TRUE;
   MM344_RivetingSupportRightInstant.CylinderNumber := 18;
   MM344_RivetingSupportRightInstant.HMICommand := 0;
   MM344_RivetingSupportRightInstant.BasicPositionCondition := TRUE;
   MM344_RivetingSupportRightInstant.WorkPositionCondition := FALSE;
   MM344_RivetingSupportRightInstant.BasicPositionSensor := TRUE;
   MM344_RivetingSupportRightInstant.WorkPositionSensor := FALSE;
   MM344_RivetingSupportRightInstant.TRIGGER := TRUE;
   MM344_RivetingSupportRightInstant.RESET := FALSE;
   MM344_RivetingSupportRightInstant.DELAY_BASIC := T#100MS;
   MM344_RivetingSupportRightInstant.DELAY_WORK := T#100MS;
   MM344_RivetingSupportRightInstant.DELAY_FREE := T#100MS;
   MM344_RivetingSupportRightInstant.ERROR_TIME := T#10S;
   MM344_RivetingSupportRightInstant.ValveDelay := T#0MS;
   MM344_RivetingSupportRightInstant.iNoCollisionBasic := TRUE;
   MM344_RivetingSupportRightInstant.iNoCollisionWork := TRUE;
   MM344_RivetingSupportRightInstant.iNoCollisionFree := TRUE;
   MM344_RivetingSupportRightInstant.VALVE_BASIC := FALSE;
   MM344_RivetingSupportRightInstant.VALVE_WORK := FALSE;
   MM344_RivetingSupportRightInstant.ERROR_BASIC := FALSE;
   MM344_RivetingSupportRightInstant.ERROR_WORK := FALSE;
   MM344_RivetingSupportRightInstant.HMIStatus := 1;
   MM344_RivetingSupportRightInstant.MOVE_BASIC := FALSE;
   MM344_RivetingSupportRightInstant.MOVE_WORK := FALSE;
   MM344_RivetingSupportRightInstant.MOVE_FREE := TRUE;
   MM344_RivetingSupportRightInstant."4l+Started" := FALSE;
   MM344_RivetingSupportRightInstant.InitCommandBP := FALSE;
   MM344_RivetingSupportRightInstant.InitCommandWP := FALSE;
   MM344_RivetingSupportRightInstant.BasicWorkStartWP := FALSE;
   MM344_RivetingSupportRightInstant.BasicWorkStartBP := FALSE;
   MM344_RivetingSupportRightInstant.work_valve := FALSE;
   MM344_RivetingSupportRightInstant.basic_valve := FALSE;
   MM344_RivetingSupportRightInstant.free_valve := FALSE;
   MM344_RivetingSupportRightInstant.baspos_error.PT := T#0MS;
   MM344_RivetingSupportRightInstant.baspos_error.IN := FALSE;
   MM344_RivetingSupportRightInstant.workpos_error.PT := T#0MS;
   MM344_RivetingSupportRightInstant.workpos_error.IN := FALSE;
   MM344_RivetingSupportRightInstant.baspos_delay.PT := T#0MS;
   MM344_RivetingSupportRightInstant.baspos_delay.IN := FALSE;
   MM344_RivetingSupportRightInstant.workpos_delay.PT := T#0MS;
   MM344_RivetingSupportRightInstant.workpos_delay.IN := FALSE;
   MM344_RivetingSupportRightInstant.CylinderOperationOld.InWp := FALSE;
   MM344_RivetingSupportRightInstant.CylinderOperationOld.InBp := FALSE;
   MM344_RivetingSupportRightInstant.CylinderOperationOld.InFp := TRUE;
   MM344_RivetingSupportRightInstant.CylinderOperationOld.ToWp := FALSE;
   MM344_RivetingSupportRightInstant.CylinderOperationOld.ToBp := FALSE;
   MM344_RivetingSupportRightInstant.CylinderOperationOld.ToFp := TRUE;
   MM344_RivetingSupportRightInstant.IEC_Timer_0_Instance.PT := T#0MS;
   MM344_RivetingSupportRightInstant.IEC_Timer_0_Instance.IN := FALSE;
   MM344_RivetingSupportRightInstant.R_TRIG_Instance.CLK := FALSE;
   MM344_RivetingSupportRightInstant.R_TRIG_Instance.Q := FALSE;
   MM344_RivetingSupportRightInstant.R_TRIG_Instance.Stat_Bit := FALSE;
   MM344_RivetingSupportRightInstant.IEC_Timer_0_Instance_1.PT := T#0MS;
   MM344_RivetingSupportRightInstant.IEC_Timer_0_Instance_1.IN := FALSE;
   MM344_RivetingSupportRightInstant.IEC_Timer_0_Instance_2.PT := T#0MS;
   MM344_RivetingSupportRightInstant.IEC_Timer_0_Instance_2.IN := FALSE;
   MM344_RivetingSupportRightInstant.IEC_Timer_0_Instance_3.PT := T#0MS;
   MM344_RivetingSupportRightInstant.IEC_Timer_0_Instance_3.IN := FALSE;
   MM344_RivetingSupportRightInstant.IEC_Timer_0_Instance_4.PT := T#0MS;
   MM344_RivetingSupportRightInstant.IEC_Timer_0_Instance_4.IN := FALSE;
END_DATA_BLOCK
